LIN {X 0,Y 231.334,Z 988.847,A -85,B 0,C 180,E1 18236.93,E2 18236.93} C_VEL
LIN {X 0,Y 220.911,Z 1008.235,A -85,B 0,C 180,E1 18251.991,E2 18251.991} C_VEL
LIN {X 0,Y 219.134,Z 1015.208,A -85,B 0,C 180,E1 18264.035,E2 18264.035} C_VEL
LIN {X 0,Y 219.137,Z 1015.4,A -85,B 0,C 180,E1 18275.961,E2 18275.961} C_VEL
LIN {X 0,Y 222.596,Z 1005.334,A -85,B 0,C 180,E1 18292.021,E2 18292.021} C_VEL
LIN {X 0,Y 238.295,Z 981.214,A -85,B 0,C 180,E1 18308.382,E2 18308.382} C_VEL
LIN {X 0,Y 267.201,Z 942.328,A -85,B 0,C 180,E1 18321.811,E2 18321.811} C_VEL
LIN {X 0,Y 301.641,Z 891.524,A -85,B 0,C 180,E1 18330.943,E2 18330.943} C_VEL
LIN {X 0,Y 323.469,Z 851.273,A -85,B 0,C 180,E1 18335.504,E2 18335.504} C_VEL
LIN {X 0,Y 324.253,Z 838.125,A -85,B 0,C 180,E1 18342.326,E2 18342.326} C_VEL
LIN {X 0,Y 323.893,Z 839.008,A -85,B 0,C 180,E1 18347.863,E2 18347.863} C_VEL
LIN {X 0,Y 321.358,Z 853.442,A -85,B 0,C 180,E1 18354.273,E2 18354.273} C_VEL
LIN {X 0,Y 299.51,Z 890.449,A -85,B 0,C 180,E1 18358.703,E2 18358.703} C_VEL
LIN {X 0,Y 278.664,Z 915.584,A -85,B 0,C 180,E1 18361.445,E2 18361.445} C_VEL
LIN {X 0,Y 245.109,Z 956.502,A -85,B 0,C 180,E1 18372.917,E2 18372.917} C_VEL
LIN {X 0,Y 221.401,Z 984.345,A -85,B 0,C 180,E1 18388.646,E2 18388.646} C_VEL
LIN {X 0,Y 212.14,Z 997.349,A -85,B 0,C 180,E1 18404.662,E2 18404.662} C_VEL
LIN {X 0,Y 209.736,Z 999.603,A -85,B 0,C 180,E1 18421.947,E2 18421.947} C_VEL
LIN {X 0,Y 214.542,Z 991.139,A -85,B 0,C 180,E1 18437.75,E2 18437.75} C_VEL
LIN {X 0,Y 229.062,Z 968.541,A -85,B 0,C 180,E1 18454.559,E2 18454.559} C_VEL
LIN {X 0,Y 254.848,Z 932.339,A -85,B 0,C 180,E1 18467.893,E2 18467.893} C_VEL
LIN {X 0,Y 284.972,Z 883.616,A -85,B 0,C 180,E1 18477.345,E2 18477.345} C_VEL
LIN {X 0,Y 301.612,Z 849.625,A -85,B 0,C 180,E1 18481.47,E2 18481.47} C_VEL
LIN {X 0,Y 294.558,Z 819.144,A -85,B 0,C 180,E1 18491.629,E2 18491.629} C_VEL
LIN {X 0,Y 285.95,Z 795.84,A -85,B 0,C 180,E1 18503.391,E2 18503.391} C_VEL
LIN {X 0,Y 280.392,Z 783.23,A -85,B 0,C 180,E1 18516.018,E2 18516.018} C_VEL
LIN {X 0,Y 280.562,Z 781.44,A -85,B 0,C 180,E1 18529.053,E2 18529.053} C_VEL
LIN {X 0,Y 284.564,Z 787.554,A -85,B 0,C 180,E1 18538.437,E2 18538.437} C_VEL
LIN {X 0,Y 293.059,Z 807.387,A -85,B 0,C 180,E1 18550.405,E2 18550.405} C_VEL
LIN {X 0,Y 302.403,Z 835.998,A -85,B 0,C 180,E1 18560.91,E2 18560.91} C_VEL
LIN {X 0,Y 304.622,Z 853.266,A -85,B 0,C 180,E1 18565.354,E2 18565.354} C_VEL
LIN {X 0,Y 275.554,Z 910.337,A -85,B 0,C 180,E1 18572.136,E2 18572.136} C_VEL
LIN {X 0,Y 245.448,Z 957.331,A -85,B 0,C 180,E1 18582.736,E2 18582.736} C_VEL
LIN {X 0,Y 222.895,Z 990.368,A -85,B 0,C 180,E1 18596.995,E2 18596.995} C_VEL
LIN {X 0,Y 212.514,Z 1009.322,A -85,B 0,C 180,E1 18613.202,E2 18613.202} C_VEL
LIN {X 0,Y 211.113,Z 1015.708,A -85,B 0,C 180,E1 18627.938,E2 18627.938} C_VEL
LIN {X 0,Y 211.662,Z 1012.771,A -85,B 0,C 180,E1 18642.419,E2 18642.419} C_VEL
LIN {X 0,Y 220.362,Z 997.045,A -85,B 0,C 180,E1 18659.951,E2 18659.951} C_VEL
LIN {X 0,Y 244.359,Z 965.515,A -85,B 0,C 180,E1 18676.299,E2 18676.299} C_VEL
LIN {X 0,Y 278.974,Z 920.137,A -85,B 0,C 180,E1 18688.065,E2 18688.065} C_VEL
LIN {X 0,Y 314.593,Z 864.629,A -85,B 0,C 180,E1 18695.39,E2 18695.39} C_VEL
LIN {X 0,Y 319.046,Z 855.506,A -85,B 0,C 180,E1 18696.616,E2 18696.616} C_VEL
LIN {X 0,Y 320.141,Z 845.375,A -85,B 0,C 180,E1 18702.091,E2 18702.091} C_VEL
LIN {X 0,Y 319.7,Z 845.822,A -85,B 0,C 180,E1 18707.701,E2 18707.701} C_VEL
LIN {X 0,Y 316.504,Z 858.344,A -85,B 0,C 180,E1 18713.297,E2 18713.297} C_VEL
LIN {X 0,Y 281.686,Z 911.578,A -85,B 0,C 180,E1 18720.654,E2 18720.654} C_VEL
LIN {X 0,Y 278.664,Z 915.584,A -85,B 0,C 180,E1 18721.445,E2 18721.445} C_VEL
LIN {X 0,Y 256.83,Z 937.989,A -85,B 0,C 180,E1 18725.038,E2 18725.038} C_VEL
LIN {X 0,Y 224.568,Z 973.616,A -85,B 0,C 180,E1 18739.578,E2 18739.578} C_VEL
LIN {X 0,Y 207.548,Z 993.263,A -85,B 0,C 180,E1 18756.625,E2 18756.625} C_VEL
LIN {X 0,Y 201.91,Z 1000.154,A -85,B 0,C 180,E1 18772.174,E2 18772.174} C_VEL
LIN {X 0,Y 203.32,Z 997.547,A -85,B 0,C 180,E1 18789.01,E2 18789.01} C_VEL
LIN {X 0,Y 212.229,Z 982.956,A -85,B 0,C 180,E1 18806.501,E2 18806.501} C_VEL
LIN {X 0,Y 234.308,Z 953.213,A -85,B 0,C 180,E1 18822.646,E2 18822.646} C_VEL
LIN {X 0,Y 263.917,Z 910.873,A -85,B 0,C 180,E1 18834.188,E2 18834.188} C_VEL
LIN {X 0,Y 293.679,Z 858.461,A -85,B 0,C 180,E1 18841.767,E2 18841.767} C_VEL
LIN {X 0,Y 295.528,Z 850.294,A -85,B 0,C 180,E1 18843.304,E2 18843.304} C_VEL
LIN {X 0,Y 288.868,Z 821.3,A -85,B 0,C 180,E1 18853.805,E2 18853.805} C_VEL
LIN {X 0,Y 281.434,Z 800.636,A -85,B 0,C 180,E1 18865.481,E2 18865.481} C_VEL
LIN {X 0,Y 277.598,Z 790.868,A -85,B 0,C 180,E1 18875.761,E2 18875.761} C_VEL
LIN {X 0,Y 277.86,Z 788.939,A -85,B 0,C 180,E1 18888.945,E2 18888.945} C_VEL
LIN {X 0,Y 281.599,Z 795.076,A -85,B 0,C 180,E1 18898.421,E2 18898.421} C_VEL
LIN {X 0,Y 289.554,Z 815.2,A -85,B 0,C 180,E1 18910.532,E2 18910.532} C_VEL
LIN {X 0,Y 297.985,Z 844.388,A -85,B 0,C 180,E1 18921.235,E2 18921.235} C_VEL
LIN {X 0,Y 299.184,Z 855.972,A -85,B 0,C 180,E1 18924.294,E2 18924.294} C_VEL
LIN {X 0,Y 269.29,Z 912.298,A -85,B 0,C 180,E1 18931.138,E2 18931.138} C_VEL
LIN {X 0,Y 237.95,Z 959.184,A -85,B 0,C 180,E1 18942.085,E2 18942.085} C_VEL
LIN {X 0,Y 213.687,Z 993.04,A -85,B 0,C 180,E1 18957.813,E2 18957.813} C_VEL
LIN {X 0,Y 204.098,Z 1010.58,A -85,B 0,C 180,E1 18974.913,E2 18974.913} C_VEL
LIN {X 0,Y 203.112,Z 1015.397,A -85,B 0,C 180,E1 18987.857,E2 18987.857} C_VEL
LIN {X 0,Y 203.722,Z 1012.51,A -85,B 0,C 180,E1 19002.912,E2 19002.912} C_VEL
LIN {X 0,Y 213.178,Z 996.923,A -85,B 0,C 180,E1 19021.065,E2 19021.065} C_VEL
LIN {X 0,Y 239.023,Z 965.172,A -85,B 0,C 180,E1 19037.934,E2 19037.934} C_VEL
LIN {X 0,Y 275.499,Z 919.867,A -85,B 0,C 180,E1 19049.671,E2 19049.671} C_VEL
LIN {X 0,Y 312.833,Z 863.926,A -85,B 0,C 180,E1 19056.911,E2 19056.911} C_VEL
LIN {X 0,Y 315.38,Z 855.567,A -85,B 0,C 180,E1 19059.769,E2 19059.769} C_VEL
LIN {X 0,Y 316.057,Z 850.77,A -85,B 0,C 180,E1 19064.724,E2 19064.724} C_VEL
LIN {X 0,Y 313.716,Z 858.36,A -85,B 0,C 180,E1 19070.858,E2 19070.858} C_VEL
LIN {X 0,Y 310.109,Z 866.089,A -85,B 0,C 180,E1 19072.588,E2 19072.588} C_VEL
LIN {X 0,Y 273.08,Z 918.562,A -85,B 0,C 180,E1 19080.396,E2 19080.396} C_VEL
LIN {X 0,Y 256.83,Z 937.989,A -85,B 0,C 180,E1 19085.038,E2 19085.038} C_VEL
LIN {X 0,Y 234.754,Z 957.261,A -85,B 0,C 180,E1 19089.71,E2 19089.71} C_VEL
LIN {X 0,Y 206.942,Z 985.713,A -85,B 0,C 180,E1 19106.686,E2 19106.686} C_VEL
LIN {X 0,Y 196.73,Z 997.789,A -85,B 0,C 180,E1 19122.878,E2 19122.878} C_VEL
LIN {X 0,Y 193.391,Z 1000.578,A -85,B 0,C 180,E1 19139.334,E2 19139.334} C_VEL
LIN {X 0,Y 197.092,Z 995.113,A -85,B 0,C 180,E1 19154.396,E2 19154.396} C_VEL
LIN {X 0,Y 210.213,Z 975.921,A -85,B 0,C 180,E1 19172.796,E2 19172.796} C_VEL
LIN {X 0,Y 236.373,Z 942.604,A -85,B 0,C 180,E1 19187.758,E2 19187.758} C_VEL
LIN {X 0,Y 268.795,Z 895.644,A -85,B 0,C 180,E1 19198.361,E2 19198.361} C_VEL
LIN {X 0,Y 290.059,Z 855.543,A -85,B 0,C 180,E1 19203.794,E2 19203.794} C_VEL
LIN {X 0,Y 284.641,Z 828.293,A -85,B 0,C 180,E1 19213.929,E2 19213.929} C_VEL
LIN {X 0,Y 278.283,Z 808.54,A -85,B 0,C 180,E1 19225.034,E2 19225.034} C_VEL
LIN {X 0,Y 274.609,Z 798.301,A -85,B 0,C 180,E1 19235.766,E2 19235.766} C_VEL
LIN {X 0,Y 274.847,Z 796.329,A -85,B 0,C 180,E1 19248.823,E2 19248.823} C_VEL
LIN {X 0,Y 278.524,Z 802.579,A -85,B 0,C 180,E1 19258.403,E2 19258.403} C_VEL
LIN {X 0,Y 285.889,Z 822.963,A -85,B 0,C 180,E1 19270.669,E2 19270.669} C_VEL
LIN {X 0,Y 293.137,Z 851.47,A -85,B 0,C 180,E1 19281.205,E2 19281.205} C_VEL
LIN {X 0,Y 293.003,Z 860.497,A -85,B 0,C 180,E1 19283.349,E2 19283.349} C_VEL
LIN {X 0,Y 261.861,Z 916.194,A -85,B 0,C 180,E1 19290.447,E2 19290.447} C_VEL
LIN {X 0,Y 230.34,Z 961.065,A -85,B 0,C 180,E1 19301.456,E2 19301.456} C_VEL
LIN {X 0,Y 205.706,Z 993.851,A -85,B 0,C 180,E1 19317.53,E2 19317.53} C_VEL
LIN {X 0,Y 196.04,Z 1010.665,A -85,B 0,C 180,E1 19335.132,E2 19335.132} C_VEL
LIN {X 0,Y 195.102,Z 1015.084,A -85,B 0,C 180,E1 19347.769,E2 19347.769} C_VEL
LIN {X 0,Y 195.489,Z 1013.207,A -85,B 0,C 180,E1 19361.189,E2 19361.189} C_VEL
LIN {X 0,Y 204.554,Z 998.694,A -85,B 0,C 180,E1 19380.637,E2 19380.637} C_VEL
LIN {X 0,Y 231.069,Z 968.126,A -85,B 0,C 180,E1 19398.335,E2 19398.335} C_VEL
LIN {X 0,Y 268.675,Z 924.229,A -85,B 0,C 180,E1 19410.484,E2 19410.484} C_VEL
LIN {X 0,Y 308.422,Z 868.26,A -85,B 0,C 180,E1 19418.016,E2 19418.016} C_VEL
LIN {X 0,Y 310.955,Z 861.059,A -85,B 0,C 180,E1 19420.601,E2 19420.601} C_VEL
LIN {X 0,Y 311.637,Z 857.651,A -85,B 0,C 180,E1 19424.502,E2 19424.502} C_VEL
LIN {X 0,Y 309.306,Z 863.877,A -85,B 0,C 180,E1 19430.147,E2 19430.147} C_VEL
LIN {X 0,Y 304.024,Z 872.927,A -85,B 0,C 180,E1 19431.784,E2 19431.784} C_VEL
LIN {X 0,Y 265.573,Z 923.791,A -85,B 0,C 180,E1 19439.791,E2 19439.791} C_VEL
LIN {X 0,Y 234.754,Z 957.261,A -85,B 0,C 180,E1 19449.71,E2 19449.71} C_VEL
LIN {X 0,Y 213.753,Z 973.272,A -85,B 0,C 180,E1 19455.789,E2 19455.789} C_VEL
LIN {X 0,Y 192.855,Z 993.797,A -85,B 0,C 180,E1 19474.288,E2 19474.288} C_VEL
LIN {X 0,Y 185.769,Z 1000.904,A -85,B 0,C 180,E1 19492.218,E2 19492.218} C_VEL
LIN {X 0,Y 187.915,Z 997.347,A -85,B 0,C 180,E1 19511.315,E2 19511.315} C_VEL
LIN {X 0,Y 199.177,Z 981.483,A -85,B 0,C 180,E1 19530.074,E2 19530.074} C_VEL
LIN {X 0,Y 223.883,Z 951.382,A -85,B 0,C 180,E1 19546.239,E2 19546.239} C_VEL
LIN {X 0,Y 256.545,Z 907.703,A -85,B 0,C 180,E1 19557.741,E2 19557.741} C_VEL
LIN {X 0,Y 284.491,Z 860.005,A -85,B 0,C 180,E1 19564.548,E2 19564.548} C_VEL
LIN {X 0,Y 279.831,Z 833.495,A -85,B 0,C 180,E1 19574.829,E2 19574.829} C_VEL
LIN {X 0,Y 273.829,Z 813.189,A -85,B 0,C 180,E1 19587.258,E2 19587.258} C_VEL
LIN {X 0,Y 270.884,Z 804.65,A -85,B 0,C 180,E1 19598.61,E2 19598.61} C_VEL
LIN {X 0,Y 271.782,Z 803.697,A -85,B 0,C 180,E1 19608.695,E2 19608.695} C_VEL
LIN {X 0,Y 275.188,Z 809.94,A -85,B 0,C 180,E1 19618.384,E2 19618.384} C_VEL
LIN {X 0,Y 281.542,Z 828.995,A -85,B 0,C 180,E1 19630.051,E2 19630.051} C_VEL
LIN {X 0,Y 287.77,Z 856.236,A -85,B 0,C 180,E1 19640.475,E2 19640.475} C_VEL
LIN {X 0,Y 287.09,Z 864.112,A -85,B 0,C 180,E1 19642.317,E2 19642.317} C_VEL
LIN {X 0,Y 255.032,Z 919.161,A -85,B 0,C 180,E1 19649.544,E2 19649.544} C_VEL
LIN {X 0,Y 221.372,Z 964.645,A -85,B 0,C 180,E1 19661.383,E2 19661.383} C_VEL
LIN {X 0,Y 197.966,Z 994.244,A -85,B 0,C 180,E1 19676.961,E2 19676.961} C_VEL
LIN {X 0,Y 188.343,Z 1009.805,A -85,B 0,C 180,E1 19693.617,E2 19693.617} C_VEL
LIN {X 0,Y 187.101,Z 1014.772,A -85,B 0,C 180,E1 19707.674,E2 19707.674} C_VEL
LIN {X 0,Y 187.794,Z 1012.243,A -85,B 0,C 180,E1 19723.426,E2 19723.426} C_VEL
LIN {X 0,Y 198.733,Z 997.113,A -85,B 0,C 180,E1 19743.214,E2 19743.214} C_VEL
LIN {X 0,Y 228.688,Z 965.09,A -85,B 0,C 180,E1 19761.218,E2 19761.218} C_VEL
LIN {X 0,Y 268.565,Z 920.5,A -85,B 0,C 180,E1 19772.833,E2 19772.833} C_VEL
LIN {X 0,Y 305.757,Z 869.649,A -85,B 0,C 180,E1 19779.653,E2 19779.653} C_VEL
LIN {X 0,Y 307.096,Z 864.294,A -85,B 0,C 180,E1 19784.498,E2 19784.498} C_VEL
LIN {X 0,Y 304.96,Z 868.97,A -85,B 0,C 180,E1 19789.258,E2 19789.258} C_VEL
LIN {X 0,Y 297.61,Z 880.195,A -85,B 0,C 180,E1 19791.023,E2 19791.023} C_VEL
LIN {X 0,Y 257.04,Z 930.122,A -85,B 0,C 180,E1 19799.425,E2 19799.425} C_VEL
LIN {X 0,Y 220.352,Z 966.958,A -85,B 0,C 180,E1 19812.265,E2 19812.265} C_VEL
LIN {X 0,Y 213.753,Z 973.272,A -85,B 0,C 180,E1 19815.789,E2 19815.789} C_VEL
LIN {X 0,Y 194.068,Z 985.971,A -85,B 0,C 180,E1 19823.301,E2 19823.301} C_VEL
LIN {X 0,Y 181.379,Z 998.29,A -85,B 0,C 180,E1 19840.815,E2 19840.815} C_VEL
LIN {X 0,Y 177.298,Z 1001.434,A -85,B 0,C 180,E1 19856.197,E2 19856.197} C_VEL
LIN {X 0,Y 181.076,Z 996.118,A -85,B 0,C 180,E1 19874.697,E2 19874.697} C_VEL
LIN {X 0,Y 195.447,Z 977.515,A -85,B 0,C 180,E1 19894.455,E2 19894.455} C_VEL
LIN {X 0,Y 224.171,Z 944.246,A -85,B 0,C 180,E1 19910.303,E2 19910.303} C_VEL
LIN {X 0,Y 258.34,Z 898.219,A -85,B 0,C 180,E1 19920.933,E2 19920.933} C_VEL
LIN {X 0,Y 278.842,Z 863.563,A -85,B 0,C 180,E1 19925.614,E2 19925.614} C_VEL
LIN {X 0,Y 274.781,Z 837.593,A -85,B 0,C 180,E1 19936.304,E2 19936.304} C_VEL
LIN {X 0,Y 269.524,Z 818.372,A -85,B 0,C 180,E1 19949.094,E2 19949.094} C_VEL
LIN {X 0,Y 267.535,Z 810.942,A -85,B 0,C 180,E1 19961.786,E2 19961.786} C_VEL
LIN {X 0,Y 270.733,Z 813.68,A -85,B 0,C 180,E1 19975.141,E2 19975.141} C_VEL
LIN {X 0,Y 276.265,Z 831.85,A -85,B 0,C 180,E1 19987.855,E2 19987.855} C_VEL
LIN {X 0,Y 281.999,Z 858.161,A -85,B 0,C 180,E1 19998.797,E2 19998.797} C_VEL
LIN {X 0,Y 281.654,Z 866.97,A -85,B 0,C 180,E1 20001.181,E2 20001.181} C_VEL
LIN {X 0,Y 248.416,Z 921.576,A -85,B 0,C 180,E1 20008.532,E2 20008.532} C_VEL
LIN {X 0,Y 213.941,Z 966.197,A -85,B 0,C 180,E1 20020.582,E2 20020.582} C_VEL
LIN {X 0,Y 189.581,Z 995.518,A -85,B 0,C 180,E1 20037.076,E2 20037.076} C_VEL
LIN {X 0,Y 179.86,Z 1010.863,A -85,B 0,C 180,E1 20055.722,E2 20055.722} C_VEL
LIN {X 0,Y 179.265,Z 1014.624,A -85,B 0,C 180,E1 20072.424,E2 20072.424} C_VEL
LIN {X 0,Y 182.356,Z 1007.925,A -85,B 0,C 180,E1 20091.991,E2 20091.991} C_VEL
LIN {X 0,Y 202.001,Z 986.423,A -85,B 0,C 180,E1 20112.541,E2 20112.541} C_VEL
LIN {X 0,Y 238.624,Z 950.181,A -85,B 0,C 180,E1 20127.893,E2 20127.893} C_VEL
LIN {X 0,Y 281.051,Z 902.165,A -85,B 0,C 180,E1 20137.356,E2 20137.356} C_VEL
LIN {X 0,Y 301.377,Z 874.097,A -85,B 0,C 180,E1 20140.935,E2 20140.935} C_VEL
LIN {X 0,Y 302.26,Z 871.131,A -85,B 0,C 180,E1 20144.008,E2 20144.008} C_VEL
LIN {X 0,Y 300.248,Z 874.828,A -85,B 0,C 180,E1 20148.707,E2 20148.707} C_VEL
LIN {X 0,Y 257.072,Z 927.132,A -85,B 0,C 180,E1 20156.896,E2 20156.896} C_VEL
LIN {X 0,Y 217.472,Z 965.308,A -85,B 0,C 180,E1 20169.432,E2 20169.432} C_VEL
LIN {X 0,Y 194.068,Z 985.971,A -85,B 0,C 180,E1 20183.301,E2 20183.301} C_VEL
LIN {X 0,Y 177.681,Z 995.01,A -85,B 0,C 180,E1 20192.644,E2 20192.644} C_VEL
LIN {X 0,Y 170.288,Z 1001.234,A -85,B 0,C 180,E1 20209.32,E2 20209.32} C_VEL
LIN {X 0,Y 170.976,Z 999.243,A -85,B 0,C 180,E1 20228.873,E2 20228.873} C_VEL
LIN {X 0,Y 180.284,Z 987.222,A -85,B 0,C 180,E1 20247.59,E2 20247.59} C_VEL
LIN {X 0,Y 204.97,Z 959.987,A -85,B 0,C 180,E1 20265.896,E2 20265.896} C_VEL
LIN {X 0,Y 239.725,Z 918.482,A -85,B 0,C 180,E1 20278.729,E2 20278.729} C_VEL
LIN {X 0,Y 273.111,Z 866.658,A -85,B 0,C 180,E1 20286.875,E2 20286.875} C_VEL
LIN {X 0,Y 269.766,Z 841.862,A -85,B 0,C 180,E1 20297.697,E2 20297.697} C_VEL
LIN {X 0,Y 265.842,Z 825.629,A -85,B 0,C 180,E1 20309.049,E2 20309.049} C_VEL
LIN {X 0,Y 264.085,Z 818.263,A -85,B 0,C 180,E1 20321.54,E2 20321.54} C_VEL
LIN {X 0,Y 267.167,Z 820.932,A -85,B 0,C 180,E1 20335.076,E2 20335.076} C_VEL
LIN {X 0,Y 272.113,Z 839.271,A -85,B 0,C 180,E1 20347.975,E2 20347.975} C_VEL
LIN {X 0,Y 276.785,Z 864.323,A -85,B 0,C 180,E1 20358.542,E2 20358.542} C_VEL
LIN {X 0,Y 275.65,Z 870.987,A -85,B 0,C 180,E1 20360.118,E2 20360.118} C_VEL
LIN {X 0,Y 241.565,Z 924.41,A -85,B 0,C 180,E1 20367.566,E2 20367.566} C_VEL
LIN {X 0,Y 206.832,Z 967.314,A -85,B 0,C 180,E1 20379.605,E2 20379.605} C_VEL
LIN {X 0,Y 181.322,Z 996.586,A -85,B 0,C 180,E1 20397.039,E2 20397.039} C_VEL
LIN {X 0,Y 171.63,Z 1011.484,A -85,B 0,C 180,E1 20417.227,E2 20417.227} C_VEL
LIN {X 0,Y 171.264,Z 1014.334,A -85,B 0,C 180,E1 20432.537,E2 20432.537} C_VEL
LIN {X 0,Y 173.734,Z 1009.157,A -85,B 0,C 180,E1 20450.449,E2 20450.449} C_VEL
LIN {X 0,Y 192.553,Z 989.611,A -85,B 0,C 180,E1 20472.058,E2 20472.058} C_VEL
LIN {X 0,Y 230.455,Z 954.665,A -85,B 0,C 180,E1 20488.436,E2 20488.436} C_VEL
LIN {X 0,Y 275.41,Z 906.835,A -85,B 0,C 180,E1 20498.41,E2 20498.41} C_VEL
LIN {X 0,Y 296.027,Z 880.706,A -85,B 0,C 180,E1 20501.511,E2 20501.511} C_VEL
LIN {X 0,Y 297.336,Z 877.785,A -85,B 0,C 180,E1 20503.736,E2 20503.736} C_VEL
LIN {X 0,Y 295.38,Z 880.557,A -85,B 0,C 180,E1 20507.766,E2 20507.766} C_VEL
LIN {X 0,Y 251.053,Z 931.031,A -85,B 0,C 180,E1 20515.854,E2 20515.854} C_VEL
LIN {X 0,Y 209.872,Z 968.156,A -85,B 0,C 180,E1 20528.782,E2 20528.782} C_VEL
LIN {X 0,Y 180.971,Z 992.098,A -85,B 0,C 180,E1 20548.301,E2 20548.301} C_VEL
LIN {X 0,Y 177.681,Z 995.01,A -85,B 0,C 180,E1 20552.644,E2 20552.644} C_VEL
LIN {X 0,Y 163.943,Z 1000.518,A -85,B 0,C 180,E1 20563.553,E2 20563.553} C_VEL
LIN {X 0,Y 161.896,Z 1000.774,A -85,B 0,C 180,E1 20585.053,E2 20585.053} C_VEL
LIN {X 0,Y 169.187,Z 991.814,A -85,B 0,C 180,E1 20603.565,E2 20603.565} C_VEL
LIN {X 0,Y 191.6,Z 967.799,A -85,B 0,C 180,E1 20623.748,E2 20623.748} C_VEL
LIN {X 0,Y 226.625,Z 929.183,A -85,B 0,C 180,E1 20637.955,E2 20637.955} C_VEL
LIN {X 0,Y 262.917,Z 878.68,A -85,B 0,C 180,E1 20646.79,E2 20646.79} C_VEL
LIN {X 0,Y 267.437,Z 869.992,A -85,B 0,C 180,E1 20648.118,E2 20648.118} C_VEL
LIN {X 0,Y 264.863,Z 846.938,A -85,B 0,C 180,E1 20658.744,E2 20658.744} C_VEL
LIN {X 0,Y 261.578,Z 831.468,A -85,B 0,C 180,E1 20670.416,E2 20670.416} C_VEL
LIN {X 0,Y 260.796,Z 824.922,A -85,B 0,C 180,E1 20684.783,E2 20684.783} C_VEL
LIN {X 0,Y 264.03,Z 830.528,A -85,B 0,C 180,E1 20697.272,E2 20697.272} C_VEL
LIN {X 0,Y 268.191,Z 848.196,A -85,B 0,C 180,E1 20708.912,E2 20708.912} C_VEL
LIN {X 0,Y 271.553,Z 871.209,A -85,B 0,C 180,E1 20718.559,E2 20718.559} C_VEL
LIN {X 0,Y 236.131,Z 925.362,A -85,B 0,C 180,E1 20726.177,E2 20726.177} C_VEL
LIN {X 0,Y 200.478,Z 967.64,A -85,B 0,C 180,E1 20738.242,E2 20738.242} C_VEL
LIN {X 0,Y 174.189,Z 996.225,A -85,B 0,C 180,E1 20755.737,E2 20755.737} C_VEL
LIN {X 0,Y 163.696,Z 1011.097,A -85,B 0,C 180,E1 20776.596,E2 20776.596} C_VEL
LIN {X 0,Y 163.238,Z 1014.045,A -85,B 0,C 180,E1 20792.662,E2 20792.662} C_VEL
LIN {X 0,Y 166.022,Z 1008.958,A -85,B 0,C 180,E1 20811.444,E2 20811.444} C_VEL
LIN {X 0,Y 186.464,Z 989.689,A -85,B 0,C 180,E1 20833.77,E2 20833.77} C_VEL
LIN {X 0,Y 227.416,Z 954.19,A -85,B 0,C 180,E1 20850.531,E2 20850.531} C_VEL
LIN {X 0,Y 274.407,Z 906.262,A -85,B 0,C 180,E1 20860.232,E2 20860.232} C_VEL
LIN {X 0,Y 292.081,Z 884.634,A -85,B 0,C 180,E1 20863.02,E2 20863.02} C_VEL
LIN {X 0,Y 290.823,Z 885.772,A -85,B 0,C 180,E1 20866.662,E2 20866.662} C_VEL
LIN {X 0,Y 245.291,Z 934.54,A -85,B 0,C 180,E1 20874.718,E2 20874.718} C_VEL
LIN {X 0,Y 201.905,Z 971.275,A -85,B 0,C 180,E1 20888.253,E2 20888.253} C_VEL
LIN {X 0,Y 172.177,Z 994.121,A -85,B 0,C 180,E1 20909.057,E2 20909.057} C_VEL
LIN {X 0,Y 163.943,Z 1000.518,A -85,B 0,C 180,E1 20923.553,E2 20923.553} C_VEL
LIN {X 0,Y 153.147,Z 1002.217,A -85,B 0,C 180,E1 20935.814,E2 20935.814} C_VEL
LIN {X 0,Y 157.374,Z 997.193,A -85,B 0,C 180,E1 20956.052,E2 20956.052} C_VEL
LIN {X 0,Y 173.69,Z 979.697,A -85,B 0,C 180,E1 20977.533,E2 20977.533} C_VEL
LIN {X 0,Y 207.085,Z 946.127,A -85,B 0,C 180,E1 20994.79,E2 20994.79} C_VEL
LIN {X 0,Y 245.278,Z 899.528,A -85,B 0,C 180,E1 21005.541,E2 21005.541} C_VEL
LIN {X 0,Y 261.881,Z 874.141,A -85,B 0,C 180,E1 21009.078,E2 21009.078} C_VEL
LIN {X 0,Y 259.937,Z 851.575,A -85,B 0,C 180,E1 21020.106,E2 21020.106} C_VEL
LIN {X 0,Y 257.301,Z 837.302,A -85,B 0,C 180,E1 21031.809,E2 21031.809} C_VEL
LIN {X 0,Y 257.023,Z 832.026,A -85,B 0,C 180,E1 21044.555,E2 21044.555} C_VEL
LIN {X 0,Y 259.849,Z 836.881,A -85,B 0,C 180,E1 21056.614,E2 21056.614} C_VEL
LIN {X 0,Y 263.379,Z 853.873,A -85,B 0,C 180,E1 21068.242,E2 21068.242} C_VEL
LIN {X 0,Y 265.907,Z 874.525,A -85,B 0,C 180,E1 21077.33,E2 21077.33} C_VEL
LIN {X 0,Y 228.668,Z 929.082,A -85,B 0,C 180,E1 21085.274,E2 21085.274} C_VEL
LIN {X 0,Y 190.934,Z 971.401,A -85,B 0,C 180,E1 21098.286,E2 21098.286} C_VEL
LIN {X 0,Y 164.911,Z 998.297,A -85,B 0,C 180,E1 21116.795,E2 21116.795} C_VEL
LIN {X 0,Y 155.806,Z 1010.689,A -85,B 0,C 180,E1 21135.904,E2 21135.904} C_VEL
LIN {X 0,Y 155.211,Z 1013.754,A -85,B 0,C 180,E1 21152.8,E2 21152.8} C_VEL
LIN {X 0,Y 158.367,Z 1008.771,A -85,B 0,C 180,E1 21172.536,E2 21172.536} C_VEL
LIN {X 0,Y 180.539,Z 989.796,A -85,B 0,C 180,E1 21195.599,E2 21195.599} C_VEL
LIN {X 0,Y 224.39,Z 954.076,A -85,B 0,C 180,E1 21212.578,E2 21212.578} C_VEL
LIN {X 0,Y 272.74,Z 906.901,A -85,B 0,C 180,E1 21221.914,E2 21221.914} C_VEL
LIN {X 0,Y 287.069,Z 890.322,A -85,B 0,C 180,E1 21224.218,E2 21224.218} C_VEL
LIN {X 0,Y 285.687,Z 891.829,A -85,B 0,C 180,E1 21225.621,E2 21225.621} C_VEL
LIN {X 0,Y 237.414,Z 940.054,A -85,B 0,C 180,E1 21234.017,E2 21234.017} C_VEL
LIN {X 0,Y 191.875,Z 975.721,A -85,B 0,C 180,E1 21248.651,E2 21248.651} C_VEL
LIN {X 0,Y 162.525,Z 996.445,A -85,B 0,C 180,E1 21270.965,E2 21270.965} C_VEL
LIN {X 0,Y 153.916,Z 1002.167,A -85,B 0,C 180,E1 21290.145,E2 21290.145} C_VEL
LIN {X 0,Y 153.147,Z 1002.217,A -85,B 0,C 180,E1 21295.814,E2 21295.814} C_VEL
LIN {X 0,Y 146.77,Z 1000.324,A -85,B 0,C 180,E1 21309.188,E2 21309.188} C_VEL
LIN {X 0,Y 157.429,Z 989.105,A -85,B 0,C 180,E1 21329.976,E2 21329.976} C_VEL
LIN {X 0,Y 186.783,Z 961.548,A -85,B 0,C 180,E1 21350.483,E2 21350.483} C_VEL
LIN {X 0,Y 226.05,Z 919.513,A -85,B 0,C 180,E1 21363.635,E2 21363.635} C_VEL
LIN {X 0,Y 256.267,Z 877.611,A -85,B 0,C 180,E1 21370.31,E2 21370.31} C_VEL
LIN {X 0,Y 254.9,Z 856.544,A -85,B 0,C 180,E1 21381.269,E2 21381.269} C_VEL
LIN {X 0,Y 253.05,Z 843.144,A -85,B 0,C 180,E1 21393.232,E2 21393.232} C_VEL
LIN {X 0,Y 253.05,Z 839.058,A -85,B 0,C 180,E1 21404.306,E2 21404.306} C_VEL
LIN {X 0,Y 255.802,Z 843.878,A -85,B 0,C 180,E1 21416.56,E2 21416.56} C_VEL
LIN {X 0,Y 258.763,Z 861.017,A -85,B 0,C 180,E1 21428.39,E2 21428.39} C_VEL
LIN {X 0,Y 259.779,Z 879.234,A -85,B 0,C 180,E1 21436.355,E2 21436.355} C_VEL
LIN {X 0,Y 222.765,Z 930.677,A -85,B 0,C 180,E1 21443.924,E2 21443.924} C_VEL
LIN {X 0,Y 183.578,Z 972.771,A -85,B 0,C 180,E1 21457.278,E2 21457.278} C_VEL
LIN {X 0,Y 155.941,Z 999.921,A -85,B 0,C 180,E1 21477.636,E2 21477.636} C_VEL
LIN {X 0,Y 147.115,Z 1012.091,A -85,B 0,C 180,E1 21501.096,E2 21501.096} C_VEL
LIN {X 0,Y 147.113,Z 1012.965,A -85,B 0,C 180,E1 21518.899,E2 21518.899} C_VEL
LIN {X 0,Y 156.231,Z 1003.989,A -85,B 0,C 180,E1 21542.291,E2 21542.291} C_VEL
LIN {X 0,Y 190.312,Z 978.576,A -85,B 0,C 180,E1 21564.817,E2 21564.817} C_VEL
LIN {X 0,Y 238.714,Z 939.313,A -85,B 0,C 180,E1 21578.394,E2 21578.394} C_VEL
LIN {X 0,Y 278.518,Z 899.892,A -85,B 0,C 180,E1 21584.546,E2 21584.546} C_VEL
LIN {X 0,Y 226.273,Z 947.876,A -85,B 0,C 180,E1 21593.996,E2 21593.996} C_VEL
LIN {X 0,Y 181.644,Z 979.927,A -85,B 0,C 180,E1 21609.142,E2 21609.142} C_VEL
LIN {X 0,Y 153.216,Z 998.365,A -85,B 0,C 180,E1 21632.661,E2 21632.661} C_VEL
LIN {X 0,Y 145.09,Z 1002.591,A -85,B 0,C 180,E1 21655.702,E2 21655.702} C_VEL
LIN {X 0,Y 146.77,Z 1000.324,A -85,B 0,C 180,E1 21669.188,E2 21669.188} C_VEL
LIN {X 0,Y 144.402,Z 994.947,A -85,B 0,C 180,E1 21683.079,E2 21683.079} C_VEL
LIN {X 0,Y 167.916,Z 973.548,A -85,B 0,C 180,E1 21705.734,E2 21705.734} C_VEL
LIN {X 0,Y 205.981,Z 937.39,A -85,B 0,C 180,E1 21721.215,E2 21721.215} C_VEL
LIN {X 0,Y 246.556,Z 887.777,A -85,B 0,C 180,E1 21730.592,E2 21730.592} C_VEL
LIN {X 0,Y 250.742,Z 880.052,A -85,B 0,C 180,E1 21732.046,E2 21732.046} C_VEL
LIN {X 0,Y 249.779,Z 859.678,A -85,B 0,C 180,E1 21743.76,E2 21743.76} C_VEL
LIN {X 0,Y 248.604,Z 849.213,A -85,B 0,C 180,E1 21754.533,E2 21754.533} C_VEL
LIN {X 0,Y 249.5,Z 846.162,A -85,B 0,C 180,E1 21767.67,E2 21767.67} C_VEL
LIN {X 0,Y 251.765,Z 852.591,A -85,B 0,C 180,E1 21778.233,E2 21778.233} C_VEL
LIN {X 0,Y 254.276,Z 871.775,A -85,B 0,C 180,E1 21790.444,E2 21790.444} C_VEL
LIN {X 0,Y 253.467,Z 883.768,A -85,B 0,C 180,E1 21795.169,E2 21795.169} C_VEL
LIN {X 0,Y 213.601,Z 936.151,A -85,B 0,C 180,E1 21803.363,E2 21803.363} C_VEL
LIN {X 0,Y 174.043,Z 976.122,A -85,B 0,C 180,E1 21817.308,E2 21817.308} C_VEL
LIN {X 0,Y 146.827,Z 1001.625,A -85,B 0,C 180,E1 21838.879,E2 21838.879} C_VEL
LIN {X 0,Y 139.154,Z 1011.695,A -85,B 0,C 180,E1 21860.582,E2 21860.582} C_VEL
LIN {X 0,Y 139.156,Z 1012.677,A -85,B 0,C 180,E1 21879.412,E2 21879.412} C_VEL
LIN {X 0,Y 151.117,Z 1002.583,A -85,B 0,C 180,E1 21905.966,E2 21905.966} C_VEL
LIN {X 0,Y 188.116,Z 977.188,A -85,B 0,C 180,E1 21927.89,E2 21927.89} C_VEL
LIN {X 0,Y 240.546,Z 936.436,A -85,B 0,C 180,E1 21941.031,E2 21941.031} C_VEL
LIN {X 0,Y 264.985,Z 913.838,A -85,B 0,C 180,E1 21944.824,E2 21944.824} C_VEL
LIN {X 0,Y 212.866,Z 956.758,A -85,B 0,C 180,E1 21954.528,E2 21954.528} C_VEL
LIN {X 0,Y 167.783,Z 985.938,A -85,B 0,C 180,E1 21971.561,E2 21971.561} C_VEL
LIN {X 0,Y 142.553,Z 1000.753,A -85,B 0,C 180,E1 21997.024,E2 21997.024} C_VEL
LIN {X 0,Y 137.093,Z 1002.569,A -85,B 0,C 180,E1 22020.126,E2 22020.126} C_VEL
LIN {X 0,Y 144.402,Z 994.947,A -85,B 0,C 180,E1 22043.079,E2 22043.079} C_VEL
LIN {X 0,Y 147.008,Z 986.464,A -85,B 0,C 180,E1 22056.653,E2 22056.653} C_VEL
LIN {X 0,Y 181.916,Z 956.572,A -85,B 0,C 180,E1 22076.671,E2 22076.671} C_VEL
LIN {X 0,Y 222.303,Z 914.776,A -85,B 0,C 180,E1 22088.218,E2 22088.218} C_VEL
LIN {X 0,Y 245.132,Z 885.142,A -85,B 0,C 180,E1 22092.646,E2 22092.646} C_VEL
LIN {X 0,Y 244.992,Z 866.148,A -85,B 0,C 180,E1 22103.911,E2 22103.911} C_VEL
LIN {X 0,Y 244.234,Z 855.113,A -85,B 0,C 180,E1 22116.14,E2 22116.14} C_VEL
LIN {X 0,Y 245.225,Z 852.942,A -85,B 0,C 180,E1 22127.452,E2 22127.452} C_VEL
LIN {X 0,Y 247.287,Z 859.389,A -85,B 0,C 180,E1 22138.201,E2 22138.201} C_VEL
LIN {X 0,Y 248.984,Z 877.707,A -85,B 0,C 180,E1 22150.135,E2 22150.135} C_VEL
LIN {X 0,Y 248.355,Z 886.343,A -85,B 0,C 180,E1 22153.774,E2 22153.774} C_VEL
LIN {X 0,Y 207.166,Z 938.435,A -85,B 0,C 180,E1 22162.046,E2 22162.046} C_VEL
LIN {X 0,Y 166.644,Z 977.418,A -85,B 0,C 180,E1 22176.21,E2 22176.21} C_VEL
LIN {X 0,Y 138.709,Z 1002.1,A -85,B 0,C 180,E1 22198.685,E2 22198.685} C_VEL
LIN {X 0,Y 131.169,Z 1011.288,A -85,B 0,C 180,E1 22220.003,E2 22220.003} C_VEL
LIN {X 0,Y 131.174,Z 1012.388,A -85,B 0,C 180,E1 22239.991,E2 22239.991} C_VEL
LIN {X 0,Y 142.503,Z 1003.797,A -85,B 0,C 180,E1 22265.851,E2 22265.851} C_VEL
LIN {X 0,Y 181.219,Z 979.288,A -85,B 0,C 180,E1 22289.13,E2 22289.13} C_VEL
LIN {X 0,Y 234.818,Z 940.359,A -85,B 0,C 180,E1 22302.314,E2 22302.314} C_VEL
LIN {X 0,Y 250.508,Z 927.008,A -85,B 0,C 180,E1 22304.908,E2 22304.908} C_VEL
LIN {X 0,Y 197.371,Z 966.078,A -85,B 0,C 180,E1 22315.658,E2 22315.658} C_VEL
LIN {X 0,Y 154.24,Z 991.032,A -85,B 0,C 180,E1 22334.303,E2 22334.303} C_VEL
LIN {X 0,Y 133.381,Z 1001.907,A -85,B 0,C 180,E1 22358.825,E2 22358.825} C_VEL
LIN {X 0,Y 129.766,Z 1001.904,A -85,B 0,C 180,E1 22385.841,E2 22385.841} C_VEL
LIN {X 0,Y 139.584,Z 992.684,A -85,B 0,C 180,E1 22408.445,E2 22408.445} C_VEL
LIN {X 0,Y 147.008,Z 986.464,A -85,B 0,C 180,E1 22416.653,E2 22416.653} C_VEL
LIN {X 0,Y 155.035,Z 974.872,A -85,B 0,C 180,E1 22429.055,E2 22429.055} C_VEL
LIN {X 0,Y 195.832,Z 939.301,A -85,B 0,C 180,E1 22444.683,E2 22444.683} C_VEL
LIN {X 0,Y 238.371,Z 890.346,A -85,B 0,C 180,E1 22453.788,E2 22453.788} C_VEL
LIN {X 0,Y 240.037,Z 874.97,A -85,B 0,C 180,E1 22462.216,E2 22462.216} C_VEL
LIN {X 0,Y 239.711,Z 863.121,A -85,B 0,C 180,E1 22473.747,E2 22473.747} C_VEL
LIN {X 0,Y 240.84,Z 859.656,A -85,B 0,C 180,E1 22487.614,E2 22487.614} C_VEL
LIN {X 0,Y 242.622,Z 866.026,A -85,B 0,C 180,E1 22498.167,E2 22498.167} C_VEL
LIN {X 0,Y 243.679,Z 883.624,A -85,B 0,C 180,E1 22509.814,E2 22509.814} C_VEL
LIN {X 0,Y 242.057,Z 890.754,A -85,B 0,C 180,E1 22512.535,E2 22512.535} C_VEL
LIN {X 0,Y 200.724,Z 940.611,A -85,B 0,C 180,E1 22520.665,E2 22520.665} C_VEL
LIN {X 0,Y 158.381,Z 979.41,A -85,B 0,C 180,E1 22535.461,E2 22535.461} C_VEL
LIN {X 0,Y 129.217,Z 1003.874,A -85,B 0,C 180,E1 22560.634,E2 22560.634} C_VEL
LIN {X 0,Y 122.977,Z 1012.063,A -85,B 0,C 180,E1 22586.459,E2 22586.459} C_VEL
LIN {X 0,Y 124.426,Z 1011.03,A -85,B 0,C 180,E1 22607.75,E2 22607.75} C_VEL
LIN {X 0,Y 145.543,Z 998.147,A -85,B 0,C 180,E1 22636.309,E2 22636.309} C_VEL
LIN {X 0,Y 195.012,Z 968.463,A -85,B 0,C 180,E1 22656.719,E2 22656.719} C_VEL
LIN {X 0,Y 236.214,Z 938.679,A -85,B 0,C 180,E1 22665.005,E2 22665.005} C_VEL
LIN {X 0,Y 182.746,Z 973.766,A -85,B 0,C 180,E1 22676.736,E2 22676.736} C_VEL
LIN {X 0,Y 140.379,Z 995.655,A -85,B 0,C 180,E1 22698.153,E2 22698.153} C_VEL
LIN {X 0,Y 123.641,Z 1003.05,A -85,B 0,C 180,E1 22722.558,E2 22722.558} C_VEL
LIN {X 0,Y 122.285,Z 1001.579,A -85,B 0,C 180,E1 22748.746,E2 22748.746} C_VEL
LIN {X 0,Y 134.985,Z 990.795,A -85,B 0,C 180,E1 22773.225,E2 22773.225} C_VEL
LIN {X 0,Y 155.035,Z 974.872,A -85,B 0,C 180,E1 22789.055,E2 22789.055} C_VEL
LIN {X 0,Y 168.442,Z 960.146,A -85,B 0,C 180,E1 22799.506,E2 22799.506} C_VEL
LIN {X 0,Y 212.124,Z 918.653,A -85,B 0,C 180,E1 22811.391,E2 22811.391} C_VEL
LIN {X 0,Y 234.106,Z 891.436,A -85,B 0,C 180,E1 22815.829,E2 22815.829} C_VEL
LIN {X 0,Y 234.98,Z 874.447,A -85,B 0,C 180,E1 22827.91,E2 22827.91} C_VEL
LIN {X 0,Y 235.171,Z 867.15,A -85,B 0,C 180,E1 22839.347,E2 22839.347} C_VEL
LIN {X 0,Y 237.227,Z 867.936,A -85,B 0,C 180,E1 22852.568,E2 22852.568} C_VEL
LIN {X 0,Y 238.153,Z 880.956,A -85,B 0,C 180,E1 22864.525,E2 22864.525} C_VEL
LIN {X 0,Y 237.492,Z 892.799,A -85,B 0,C 180,E1 22870.971,E2 22870.971} C_VEL
LIN {X 0,Y 194.752,Z 942.415,A -85,B 0,C 180,E1 22879.114,E2 22879.114} C_VEL
LIN {X 0,Y 153.645,Z 978.546,A -85,B 0,C 180,E1 22892.901,E2 22892.901} C_VEL
LIN {X 0,Y 123.539,Z 1001.971,A -85,B 0,C 180,E1 22916.437,E2 22916.437} C_VEL
LIN {X 0,Y 114.978,Z 1011.021,A -85,B 0,C 180,E1 22941.171,E2 22941.171} C_VEL
LIN {X 0,Y 115.268,Z 1011.816,A -85,B 0,C 180,E1 22961.386,E2 22961.386} C_VEL
LIN {X 0,Y 130.151,Z 1003.312,A -85,B 0,C 180,E1 22990.854,E2 22990.854} C_VEL
LIN {X 0,Y 176.181,Z 978.506,A -85,B 0,C 180,E1 23014.745,E2 23014.745} C_VEL
LIN {X 0,Y 221.192,Z 949.716,A -85,B 0,C 180,E1 23024.65,E2 23024.65} C_VEL
LIN {X 0,Y 164.137,Z 982.574,A -85,B 0,C 180,E1 23039.558,E2 23039.558} C_VEL
LIN {X 0,Y 125.288,Z 1000.054,A -85,B 0,C 180,E1 23065.166,E2 23065.166} C_VEL
LIN {X 0,Y 113.108,Z 1003.872,A -85,B 0,C 180,E1 23092.864,E2 23092.864} C_VEL
LIN {X 0,Y 117.777,Z 999.045,A -85,B 0,C 180,E1 23118.859,E2 23118.859} C_VEL
LIN {X 0,Y 140.334,Z 981.878,A -85,B 0,C 180,E1 23145.688,E2 23145.688} C_VEL
LIN {X 0,Y 168.442,Z 960.146,A -85,B 0,C 180,E1 23159.506,E2 23159.506} C_VEL
LIN {X 0,Y 184.614,Z 942.622,A -85,B 0,C 180,E1 23168.064,E2 23168.064} C_VEL
LIN {X 0,Y 227.781,Z 896.775,A -85,B 0,C 180,E1 23176.701,E2 23176.701} C_VEL
LIN {X 0,Y 229.707,Z 883.132,A -85,B 0,C 180,E1 23185.793,E2 23185.793} C_VEL
LIN {X 0,Y 230.119,Z 875.646,A -85,B 0,C 180,E1 23194.576,E2 23194.576} C_VEL
LIN {X 0,Y 231.366,Z 872.663,A -85,B 0,C 180,E1 23206.687,E2 23206.687} C_VEL
LIN {X 0,Y 232.775,Z 877.072,A -85,B 0,C 180,E1 23216.22,E2 23216.22} C_VEL
LIN {X 0,Y 232.637,Z 893.804,A -85,B 0,C 180,E1 23228.49,E2 23228.49} C_VEL
LIN {X 0,Y 230.101,Z 898.59,A -85,B 0,C 180,E1 23229.778,E2 23229.778} C_VEL
LIN {X 0,Y 185.761,Z 947.204,A -85,B 0,C 180,E1 23238.241,E2 23238.241} C_VEL
LIN {X 0,Y 141.67,Z 983.277,A -85,B 0,C 180,E1 23253.926,E2 23253.926} C_VEL
LIN {X 0,Y 112.094,Z 1005.073,A -85,B 0,C 180,E1 23281.711,E2 23281.711} C_VEL
LIN {X 0,Y 106.965,Z 1011.315,A -85,B 0,C 180,E1 23305.928,E2 23305.928} C_VEL
LIN {X 0,Y 108.961,Z 1010.559,A -85,B 0,C 180,E1 23330.373,E2 23330.373} C_VEL
LIN {X 0,Y 135.733,Z 997.804,A -85,B 0,C 180,E1 23362.158,E2 23362.158} C_VEL
LIN {X 0,Y 193,Z 967.642,A -85,B 0,C 180,E1 23382.085,E2 23382.085} C_VEL
LIN {X 0,Y 207.053,Z 958.906,A -85,B 0,C 180,E1 23385.19,E2 23385.19} C_VEL
LIN {X 0,Y 149.433,Z 988.36,A -85,B 0,C 180,E1 23401.369,E2 23401.369} C_VEL
LIN {X 0,Y 113.596,Z 1002.289,A -85,B 0,C 180,E1 23429.737,E2 23429.737} C_VEL
LIN {X 0,Y 104.828,Z 1003.7,A -85,B 0,C 180,E1 23459.56,E2 23459.56} C_VEL
LIN {X 0,Y 114.062,Z 996.267,A -85,B 0,C 180,E1 23487.654,E2 23487.654} C_VEL
LIN {X 0,Y 143.499,Z 975.526,A -85,B 0,C 180,E1 23513.368,E2 23513.368} C_VEL
LIN {X 0,Y 184.614,Z 942.622,A -85,B 0,C 180,E1 23528.064,E2 23528.064} C_VEL
LIN {X 0,Y 202.517,Z 922.303,A -85,B 0,C 180,E1 23534.864,E2 23534.864} C_VEL
LIN {X 0,Y 223.079,Z 899.214,A -85,B 0,C 180,E1 23538.47,E2 23538.47} C_VEL
LIN {X 0,Y 224.896,Z 884.408,A -85,B 0,C 180,E1 23550.904,E2 23550.904} C_VEL
LIN {X 0,Y 225.841,Z 879.303,A -85,B 0,C 180,E1 23562.357,E2 23562.357} C_VEL
LIN {X 0,Y 227.871,Z 881.632,A -85,B 0,C 180,E1 23574.224,E2 23574.224} C_VEL
LIN {X 0,Y 227.206,Z 896.397,A -85,B 0,C 180,E1 23586.372,E2 23586.372} C_VEL
LIN {X 0,Y 225.048,Z 901.35,A -85,B 0,C 180,E1 23588.201,E2 23588.201} C_VEL
LIN {X 0,Y 180.007,Z 948.779,A -85,B 0,C 180,E1 23596.496,E2 23596.496} C_VEL
LIN {X 0,Y 134.643,Z 984.165,A -85,B 0,C 180,E1 23612.285,E2 23612.285} C_VEL
LIN {X 0,Y 104.935,Z 1004.526,A -85,B 0,C 180,E1 23639.586,E2 23639.586} C_VEL
LIN {X 0,Y 98.967,Z 1010.935,A -85,B 0,C 180,E1 23665.599,E2 23665.599} C_VEL
LIN {X 0,Y 101.319,Z 1010.333,A -85,B 0,C 180,E1 23691.987,E2 23691.987} C_VEL
LIN {X 0,Y 130.797,Z 997.906,A -85,B 0,C 180,E1 23725.035,E2 23725.035} C_VEL
LIN {X 0,Y 190.105,Z 968.733,A -85,B 0,C 180,E1 23744.306,E2 23744.306} C_VEL
LIN {X 0,Y 193.15,Z 967.04,A -85,B 0,C 180,E1 23745.143,E2 23745.143} C_VEL
LIN {X 0,Y 134.86,Z 993.243,A -85,B 0,C 180,E1 23763.299,E2 23763.299} C_VEL
LIN {X 0,Y 102.067,Z 1003.873,A -85,B 0,C 180,E1 23795.144,E2 23795.144} C_VEL
LIN {X 0,Y 97.611,Z 1002.959,A -85,B 0,C 180,E1 23827.132,E2 23827.132} C_VEL
LIN {X 0,Y 109.911,Z 994.322,A -85,B 0,C 180,E1 23853.962,E2 23853.962} C_VEL
LIN {X 0,Y 145.717,Z 970.559,A -85,B 0,C 180,E1 23879.236,E2 23879.236} C_VEL
LIN {X 0,Y 192.287,Z 932.363,A -85,B 0,C 180,E1 23892.902,E2 23892.902} C_VEL
LIN {X 0,Y 202.517,Z 922.303,A -85,B 0,C 180,E1 23894.864,E2 23894.864} C_VEL
LIN {X 0,Y 213.226,Z 907.916,A -85,B 0,C 180,E1 23899.262,E2 23899.262} C_VEL
LIN {X 0,Y 217.626,Z 902.65,A -85,B 0,C 180,E1 23900.117,E2 23900.117} C_VEL
LIN {X 0,Y 219.764,Z 890.145,A -85,B 0,C 180,E1 23911.568,E2 23911.568} C_VEL
LIN {X 0,Y 221.355,Z 885.306,A -85,B 0,C 180,E1 23926.073,E2 23926.073} C_VEL
LIN {X 0,Y 222.531,Z 889.555,A -85,B 0,C 180,E1 23936.045,E2 23936.045} C_VEL
LIN {X 0,Y 221.432,Z 902.488,A -85,B 0,C 180,E1 23946.386,E2 23946.386} C_VEL
LIN {X 0,Y 174.391,Z 950.32,A -85,B 0,C 180,E1 23954.627,E2 23954.627} C_VEL
LIN {X 0,Y 127.85,Z 984.85,A -85,B 0,C 180,E1 23970.404,E2 23970.404} C_VEL
LIN {X 0,Y 96.591,Z 1004.861,A -85,B 0,C 180,E1 23999.553,E2 23999.553} C_VEL
LIN {X 0,Y 90.939,Z 1010.548,A -85,B 0,C 180,E1 24025.209,E2 24025.209} C_VEL
LIN {X 0,Y 93.759,Z 1010.112,A -85,B 0,C 180,E1 24053.865,E2 24053.865} C_VEL
LIN {X 0,Y 126.033,Z 998.093,A -85,B 0,C 180,E1 24088.046,E2 24088.046} C_VEL
LIN {X 0,Y 178.179,Z 974.77,A -85,B 0,C 180,E1 24105.258,E2 24105.258} C_VEL
LIN {X 0,Y 118.887,Z 997.807,A -85,B 0,C 180,E1 24126.645,E2 24126.645} C_VEL
LIN {X 0,Y 94.047,Z 1004.394,A -85,B 0,C 180,E1 24154.507,E2 24154.507} C_VEL
LIN {X 0,Y 89.846,Z 1003.008,A -85,B 0,C 180,E1 24188.549,E2 24188.549} C_VEL
LIN {X 0,Y 104.816,Z 993.418,A -85,B 0,C 180,E1 24218.329,E2 24218.329} C_VEL
LIN {X 0,Y 144.135,Z 968.579,A -85,B 0,C 180,E1 24242.991,E2 24242.991} C_VEL
LIN {X 0,Y 191.366,Z 930.495,A -85,B 0,C 180,E1 24255.542,E2 24255.542} C_VEL
LIN {X 0,Y 213.226,Z 907.916,A -85,B 0,C 180,E1 24259.262,E2 24259.262} C_VEL
LIN {X 0,Y 214.751,Z 903.581,A -85,B 0,C 180,E1 24261.871,E2 24261.871} C_VEL
LIN {X 0,Y 213.167,Z 901.805,A -85,B 0,C 180,E1 24265.502,E2 24265.502} C_VEL
LIN {X 0,Y 214.861,Z 893.217,A -85,B 0,C 180,E1 24277.096,E2 24277.096} C_VEL
LIN {X 0,Y 216.985,Z 892.016,A -85,B 0,C 180,E1 24289.886,E2 24289.886} C_VEL
LIN {X 0,Y 216.74,Z 899.951,A -85,B 0,C 180,E1 24300.164,E2 24300.164} C_VEL
LIN {X 0,Y 215.355,Z 906.718,A -85,B 0,C 180,E1 24304.856,E2 24304.856} C_VEL
LIN {X 0,Y 165.563,Z 954.648,A -85,B 0,C 180,E1 24313.395,E2 24313.395} C_VEL
LIN {X 0,Y 115.602,Z 988.988,A -85,B 0,C 180,E1 24331.421,E2 24331.421} C_VEL
LIN {X 0,Y 86.381,Z 1006.438,A -85,B 0,C 180,E1 24363.941,E2 24363.941} C_VEL
LIN {X 0,Y 82.995,Z 1010.81,A -85,B 0,C 180,E1 24395.241,E2 24395.241} C_VEL
LIN {X 0,Y 97.757,Z 1006.374,A -85,B 0,C 180,E1 24434.308,E2 24434.308} C_VEL
LIN {X 0,Y 151.639,Z 986.732,A -85,B 0,C 180,E1 24461.935,E2 24461.935} C_VEL
LIN {X 0,Y 163.327,Z 981.528,A -85,B 0,C 180,E1 24465.382,E2 24465.382} C_VEL
LIN {X 0,Y 104.951,Z 1000.941,A -85,B 0,C 180,E1 24489.763,E2 24489.763} C_VEL
LIN {X 0,Y 83.71,Z 1005.113,A -85,B 0,C 180,E1 24519.529,E2 24519.529} C_VEL
LIN {X 0,Y 85.05,Z 1001.222,A -85,B 0,C 180,E1 24559.489,E2 24559.489} C_VEL
LIN {X 0,Y 111.329,Z 986.213,A -85,B 0,C 180,E1 24592.02,E2 24592.02} C_VEL
LIN {X 0,Y 158.174,Z 955.902,A -85,B 0,C 180,E1 24611.274,E2 24611.274} C_VEL
LIN {X 0,Y 207.453,Z 911.714,A -85,B 0,C 180,E1 24620.85,E2 24620.85} C_VEL
LIN {X 0,Y 211.574,Z 907.134,A -85,B 0,C 180,E1 24621.447,E2 24621.447} C_VEL
LIN {X 0,Y 213.167,Z 901.805,A -85,B 0,C 180,E1 24625.502,E2 24625.502} C_VEL
LIN {X 0,Y 209.259,Z 900.061,A -85,B 0,C 180,E1 24635.163,E2 24635.163} C_VEL
LIN {X 0,Y 211.56,Z 897.927,A -85,B 0,C 180,E1 24649.623,E2 24649.623} C_VEL
LIN {X 0,Y 211.083,Z 905.842,A -85,B 0,C 180,E1 24660.053,E2 24660.053} C_VEL
LIN {X 0,Y 209.625,Z 910.425,A -85,B 0,C 180,E1 24663.215,E2 24663.215} C_VEL
LIN {X 0,Y 160.509,Z 955.767,A -85,B 0,C 180,E1 24671.191,E2 24671.191} C_VEL
LIN {X 0,Y 111.452,Z 988.076,A -85,B 0,C 180,E1 24687.731,E2 24687.731} C_VEL
LIN {X 0,Y 79.089,Z 1005.912,A -85,B 0,C 180,E1 24721.328,E2 24721.328} C_VEL
LIN {X 0,Y 74.961,Z 1010.474,A -85,B 0,C 180,E1 24755.804,E2 24755.804} C_VEL
LIN {X 0,Y 91.998,Z 1006.33,A -85,B 0,C 180,E1 24797.922,E2 24797.922} C_VEL
LIN {X 0,Y 148.971,Z 987.266,A -85,B 0,C 180,E1 24825.405,E2 24825.405} C_VEL
LIN {X 0,Y 99.285,Z 1001.633,A -85,B 0,C 180,E1 24846.554,E2 24846.554} C_VEL
LIN {X 0,Y 73.685,Z 1005.403,A -85,B 0,C 180,E1 24886.307,E2 24886.307} C_VEL
LIN {X 0,Y 81.318,Z 999.329,A -85,B 0,C 180,E1 24929.546,E2 24929.546} C_VEL
LIN {X 0,Y 115.961,Z 980.791,A -85,B 0,C 180,E1 24960.869,E2 24960.869} C_VEL
LIN {X 0,Y 165.824,Z 947.691,A -85,B 0,C 180,E1 24976.436,E2 24976.436} C_VEL
LIN {X 0,Y 206.615,Z 910.328,A -85,B 0,C 180,E1 24983.207,E2 24983.207} C_VEL
LIN {X 0,Y 209.259,Z 900.061,A -85,B 0,C 180,E1 24995.163,E2 24995.163} C_VEL
LIN {X 0,Y 205.223,Z 903.514,A -85,B 0,C 180,E1 25004.92,E2 25004.92} C_VEL
LIN {X 0,Y 206.069,Z 907.31,A -85,B 0,C 180,E1 25015.729,E2 25015.729} C_VEL
LIN {X 0,Y 204.031,Z 914.112,A -85,B 0,C 180,E1 25021.473,E2 25021.473} C_VEL
LIN {X 0,Y 153.077,Z 958.775,A -85,B 0,C 180,E1 25029.398,E2 25029.398} C_VEL
LIN {X 0,Y 102.515,Z 989.932,A -85,B 0,C 180,E1 25046.485,E2 25046.485} C_VEL
LIN {X 0,Y 69.786,Z 1006.626,A -85,B 0,C 180,E1 25084.213,E2 25084.213} C_VEL
LIN {X 0,Y 66.951,Z 1010.138,A -85,B 0,C 180,E1 25116.502,E2 25116.502} C_VEL
LIN {X 0,Y 87.573,Z 1006.05,A -85,B 0,C 180,E1 25162.816,E2 25162.816} C_VEL
LIN {X 0,Y 134.611,Z 992.245,A -85,B 0,C 180,E1 25185.449,E2 25185.449} C_VEL
LIN {X 0,Y 79.225,Z 1004.905,A -85,B 0,C 180,E1 25216.827,E2 25216.827} C_VEL
LIN {X 0,Y 64.567,Z 1005.161,A -85,B 0,C 180,E1 25255.604,E2 25255.604} C_VEL
LIN {X 0,Y 76.273,Z 998.421,A -85,B 0,C 180,E1 25295.715,E2 25295.715} C_VEL
LIN {X 0,Y 115.868,Z 978.602,A -85,B 0,C 180,E1 25326.118,E2 25326.118} C_VEL
LIN {X 0,Y 168.27,Z 943.686,A -85,B 0,C 180,E1 25340.053,E2 25340.053} C_VEL
LIN {X 0,Y 201.368,Z 913.355,A -85,B 0,C 180,E1 25345.531,E2 25345.531} C_VEL
LIN {X 0,Y 203.762,Z 905.61,A -85,B 0,C 180,E1 25355.771,E2 25355.771} C_VEL
LIN {X 0,Y 205.223,Z 903.514,A -85,B 0,C 180,E1 25364.92,E2 25364.92} C_VEL
LIN {X 0,Y 201.638,Z 909.609,A -85,B 0,C 180,E1 25372.15,E2 25372.15} C_VEL
LIN {X 0,Y 200.457,Z 912.183,A -85,B 0,C 180,E1 25374.633,E2 25374.633} C_VEL
LIN {X 0,Y 198.318,Z 917.847,A -85,B 0,C 180,E1 25379.679,E2 25379.679} C_VEL
LIN {X 0,Y 145.412,Z 961.98,A -85,B 0,C 180,E1 25387.469,E2 25387.469} C_VEL
LIN {X 0,Y 92.523,Z 992.16,A -85,B 0,C 180,E1 25405.551,E2 25405.551} C_VEL
LIN {X 0,Y 60.602,Z 1007.287,A -85,B 0,C 180,E1 25447.93,E2 25447.93} C_VEL
LIN {X 0,Y 58.926,Z 1009.797,A -85,B 0,C 180,E1 25477.392,E2 25477.392} C_VEL
LIN {X 0,Y 81.804,Z 1006.185,A -85,B 0,C 180,E1 25526.588,E2 25526.588} C_VEL
LIN {X 0,Y 119.367,Z 996.715,A -85,B 0,C 180,E1 25545.696,E2 25545.696} C_VEL
LIN {X 0,Y 67.624,Z 1005.865,A -85,B 0,C 180,E1 25579.824,E2 25579.824} C_VEL
LIN {X 0,Y 57.282,Z 1004.26,A -85,B 0,C 180,E1 25628.451,E2 25628.451} C_VEL
LIN {X 0,Y 78.687,Z 994.607,A -85,B 0,C 180,E1 25669.999,E2 25669.999} C_VEL
LIN {X 0,Y 127.535,Z 970.003,A -85,B 0,C 180,E1 25694.555,E2 25694.555} C_VEL
LIN {X 0,Y 180.909,Z 931.52,A -85,B 0,C 180,E1 25704.879,E2 25704.879} C_VEL
LIN {X 0,Y 195.843,Z 917.328,A -85,B 0,C 180,E1 25707.144,E2 25707.144} C_VEL
LIN {X 0,Y 198.635,Z 910.059,A -85,B 0,C 180,E1 25719.842,E2 25719.842} C_VEL
LIN {X 0,Y 200.417,Z 909.47,A -85,B 0,C 180,E1 25729.039,E2 25729.039} C_VEL
LIN {X 0,Y 200.457,Z 912.183,A -85,B 0,C 180,E1 25734.633,E2 25734.633} C_VEL
LIN {X 0,Y 193.557,Z 920.618,A -85,B 0,C 180,E1 25737.513,E2 25737.513} C_VEL
LIN {X 0,Y 186.74,Z 927.187,A -85,B 0,C 180,E1 25738.408,E2 25738.408} C_VEL
LIN {X 0,Y 132.266,Z 968.487,A -85,B 0,C 180,E1 25746.502,E2 25746.502} C_VEL
LIN {X 0,Y 77.282,Z 996.428,A -85,B 0,C 180,E1 25767.901,E2 25767.901} C_VEL
LIN {X 0,Y 53.165,Z 1006.758,A -85,B 0,C 180,E1 25804.64,E2 25804.64} C_VEL
LIN {X 0,Y 50.923,Z 1009.433,A -85,B 0,C 180,E1 25838.562,E2 25838.562} C_VEL
LIN {X 0,Y 77.541,Z 1006.096,A -85,B 0,C 180,E1 25891.718,E2 25891.718} C_VEL
LIN {X 0,Y 103.992,Z 1000.438,A -85,B 0,C 180,E1 25905.863,E2 25905.863} C_VEL
LIN {X 0,Y 55.894,Z 1006.461,A -85,B 0,C 180,E1 25944.224,E2 25944.224} C_VEL
LIN {X 0,Y 53.472,Z 1002.553,A -85,B 0,C 180,E1 26005.122,E2 26005.122} C_VEL
LIN {X 0,Y 87.477,Z 988.798,A -85,B 0,C 180,E1 26044.326,E2 26044.326} C_VEL
LIN {X 0,Y 144.15,Z 958.102,A -85,B 0,C 180,E1 26062.152,E2 26062.152} C_VEL
LIN {X 0,Y 190.31,Z 921.464,A -85,B 0,C 180,E1 26068.726,E2 26068.726} C_VEL
LIN {X 0,Y 192.69,Z 915.914,A -85,B 0,C 180,E1 26079.192,E2 26079.192} C_VEL
LIN {X 0,Y 194.647,Z 915.115,A -85,B 0,C 180,E1 26088.71,E2 26088.71} C_VEL
LIN {X 0,Y 193.614,Z 920.629,A -85,B 0,C 180,E1 26097.702,E2 26097.702} C_VEL
LIN {X 0,Y 186.74,Z 927.187,A -85,B 0,C 180,E1 26098.408,E2 26098.408} C_VEL
LIN {X 0,Y 158.641,Z 948.849,A -85,B 0,C 180,E1 26098.826,E2 26098.826} C_VEL
LIN {X 0,Y 102.612,Z 982.964,A -85,B 0,C 180,E1 26109.573,E2 26109.573} C_VEL
LIN {X 0,Y 52.693,Z 1003.51,A -85,B 0,C 180,E1 26143.934,E2 26143.934} C_VEL
LIN {X 0,Y 42.927,Z 1008.023,A -85,B 0,C 180,E1 26179.809,E2 26179.809} C_VEL
LIN {X 0,Y 49.475,Z 1008.98,A -85,B 0,C 180,E1 26230.261,E2 26230.261} C_VEL
LIN {X 0,Y 89.983,Z 1003.196,A -85,B 0,C 180,E1 26265.465,E2 26265.465} C_VEL
LIN {X 0,Y 44.132,Z 1006.633,A -85,B 0,C 180,E1 26311.31,E2 26311.31} C_VEL
LIN {X 0,Y 50.603,Z 1001.129,A -85,B 0,C 180,E1 26378.632,E2 26378.632} C_VEL
LIN {X 0,Y 95.421,Z 983.667,A -85,B 0,C 180,E1 26414.164,E2 26414.164} C_VEL
LIN {X 0,Y 153.763,Z 950.252,A -85,B 0,C 180,E1 26427.032,E2 26427.032} C_VEL
LIN {X 0,Y 184.791,Z 925.277,A -85,B 0,C 180,E1 26430.779,E2 26430.779} C_VEL
LIN {X 0,Y 187.644,Z 920.594,A -85,B 0,C 180,E1 26443.505,E2 26443.505} C_VEL
LIN {X 0,Y 188.968,Z 922.107,A -85,B 0,C 180,E1 26453.029,E2 26453.029} C_VEL
LIN {X 0,Y 187.125,Z 925.279,A -85,B 0,C 180,E1 26455.807,E2 26455.807} C_VEL
LIN {X 0,Y 158.641,Z 948.849,A -85,B 0,C 180,E1 26458.826,E2 26458.826} C_VEL
LIN {X 0,Y 128.436,Z 967.511,A -85,B 0,C 180,E1 26459.573,E2 26459.573} C_VEL
LIN {X 0,Y 71.021,Z 994.719,A -85,B 0,C 180,E1 26475.916,E2 26475.916} C_VEL
LIN {X 0,Y 39.044,Z 1005.591,A -85,B 0,C 180,E1 26514.323,E2 26514.323} C_VEL
LIN {X 0,Y 35.013,Z 1008.58,A -85,B 0,C 180,E1 26562.505,E2 26562.505} C_VEL
LIN {X 0,Y 71.174,Z 1005.954,A -85,B 0,C 180,E1 26623.617,E2 26623.617} C_VEL
LIN {X 0,Y 73.027,Z 1005.613,A -85,B 0,C 180,E1 26626.244,E2 26626.244} C_VEL
LIN {X 0,Y 32.943,Z 1006.289,A -85,B 0,C 180,E1 26684.121,E2 26684.121} C_VEL
LIN {X 0,Y 47.317,Z 1000.28,A -85,B 0,C 180,E1 26749.307,E2 26749.307} C_VEL
LIN {X 0,Y 98.383,Z 981.101,A -85,B 0,C 180,E1 26780.474,E2 26780.474} C_VEL
LIN {X 0,Y 155.479,Z 947.963,A -85,B 0,C 180,E1 26790.364,E2 26790.364} C_VEL
LIN {X 0,Y 179.232,Z 929.257,A -85,B 0,C 180,E1 26792.76,E2 26792.76} C_VEL
LIN {X 0,Y 182.609,Z 925.913,A -85,B 0,C 180,E1 26807.955,E2 26807.955} C_VEL
LIN {X 0,Y 181.746,Z 928.704,A -85,B 0,C 180,E1 26813.692,E2 26813.692} C_VEL
LIN {X 0,Y 128.436,Z 967.511,A -85,B 0,C 180,E1 26819.573,E2 26819.573} C_VEL
LIN {X 0,Y 96.524,Z 982.814,A -85,B 0,C 180,E1 26821.059,E2 26821.059} C_VEL
LIN {X 0,Y 38.543,Z 1003.425,A -85,B 0,C 180,E1 26853.993,E2 26853.993} C_VEL
LIN {X 0,Y 27.156,Z 1008.147,A -85,B 0,C 180,E1 26926.21,E2 26926.21} C_VEL
LIN {X 0,Y 58.798,Z 1007.017,A -85,B 0,C 180,E1 26985.567,E2 26985.567} C_VEL
LIN {X 0,Y 26.564,Z 1006.775,A -85,B 0,C 180,E1 27031.054,E2 27031.054} C_VEL
LIN {X 0,Y 43.465,Z 999.958,A -85,B 0,C 180,E1 27118.752,E2 27118.752} C_VEL
LIN {X 0,Y 100.69,Z 979.23,A -85,B 0,C 180,E1 27145.999,E2 27145.999} C_VEL
LIN {X 0,Y 160.567,Z 943.555,A -85,B 0,C 180,E1 27153.888,E2 27153.888} C_VEL
LIN {X 0,Y 173.593,Z 933.342,A -85,B 0,C 180,E1 27155.184,E2 27155.184} C_VEL
LIN {X 0,Y 176.455,Z 931.483,A -85,B 0,C 180,E1 27169.28,E2 27169.28} C_VEL
LIN {X 0,Y 175.285,Z 933.221,A -85,B 0,C 180,E1 27171.535,E2 27171.535} C_VEL
LIN {X 0,Y 116.436,Z 972.975,A -85,B 0,C 180,E1 27177.455,E2 27177.455} C_VEL
LIN {X 0,Y 96.524,Z 982.814,A -85,B 0,C 180,E1 27181.059,E2 27181.059} C_VEL
LIN {X 0,Y 63.163,Z 994.61,A -85,B 0,C 180,E1 27183.987,E2 27183.987} C_VEL
LIN {X 0,Y 19.52,Z 1006.476,A -85,B 0,C 180,E1 27247.103,E2 27247.103} C_VEL
LIN {X 0,Y 27.363,Z 1008.142,A -85,B 0,C 180,E1 27326.269,E2 27326.269} C_VEL
LIN {X 0,Y 41.181,Z 1007.833,A -85,B 0,C 180,E1 27346.017,E2 27346.017} C_VEL
LIN {X 0,Y 24.434,Z 1003.466,A -85,B 0,C 180,E1 27468.11,E2 27468.11} C_VEL
LIN {X 0,Y 70.285,Z 990.884,A -85,B 0,C 180,E1 27504.077,E2 27504.077} C_VEL
LIN {X 0,Y 132.444,Z 961.825,A -85,B 0,C 180,E1 27514.475,E2 27514.475} C_VEL
LIN {X 0,Y 167.226,Z 937.959,A -85,B 0,C 180,E1 27517.251,E2 27517.251} C_VEL
LIN {X 0,Y 170.221,Z 936.472,A -85,B 0,C 180,E1 27529.032,E2 27529.032} C_VEL
LIN {X 0,Y 110.66,Z 975.025,A -85,B 0,C 180,E1 27534.079,E2 27534.079} C_VEL
LIN {X 0,Y 63.163,Z 994.61,A -85,B 0,C 180,E1 27543.987,E2 27543.987} C_VEL
LIN {X 0,Y 29.005,Z 1002.691,A -85,B 0,C 180,E1 27551.784,E2 27551.784} C_VEL
LIN {X 0,Y 12.429,Z 1007.259,A -85,B 0,C 180,E1 27667.585,E2 27667.585} C_VEL
LIN {X 0,Y 23.624,Z 1007.758,A -85,B 0,C 180,E1 27704.426,E2 27704.426} C_VEL
LIN {X 0,Y 31.37,Z 1001.251,A -85,B 0,C 180,E1 27856.542,E2 27856.542} C_VEL
LIN {X 0,Y 92.499,Z 981.86,A -85,B 0,C 180,E1 27874.48,E2 27874.48} C_VEL
LIN {X 0,Y 152.174,Z 948.868,A -85,B 0,C 180,E1 27879.225,E2 27879.225} C_VEL
LIN {X 0,Y 160.917,Z 942.653,A -85,B 0,C 180,E1 27879.709,E2 27879.709} C_VEL
LIN {X 0,Y 163.435,Z 941.163,A -85,B 0,C 180,E1 27886.517,E2 27886.517} C_VEL
LIN {X 0,Y 103.886,Z 977.498,A -85,B 0,C 180,E1 27890.444,E2 27890.444} C_VEL
LIN {X 0,Y 45.05,Z 998.945,A -85,B 0,C 180,E1 27901.891,E2 27901.891} C_VEL
LIN {X 0,Y 29.005,Z 1002.691,A -85,B 0,C 180,E1 27911.784,E2 27911.784} C_VEL
LIN {X 0,Y 5.278,Z 1005.678,A -85,B 0,C 180,E1 27921.156,E2 27921.156} C_VEL
LIN {X 0,Y 0.418,Z 1006.098,A -85,B 0,C 180,E1 28045.457,E2 28045.457} C_VEL
LIN {X 0,Y 42.298,Z 998.506,A -85,B 0,C 180,E1 27873.783,E2 27873.783} C_VEL
LIN {X 0,Y 107.616,Z 974.932,A -85,B 0,C 180,E1 27880.341,E2 27880.341} C_VEL
LIN {X 0,Y 155.352,Z 946.621,A -85,B 0,C 180,E1 27882.363,E2 27882.363} C_VEL
LIN {X 0,Y 156.144,Z 946.174,A -85,B 0,C 180,E1 27883.882,E2 27883.882} C_VEL
LIN {X 0,Y 94.369,Z 981.34,A -85,B 0,C 180,E1 27886.557,E2 27886.557} C_VEL
LIN {X 0,Y 30.486,Z 1001.572,A -85,B 0,C 180,E1 27894.76,E2 27894.76} C_VEL
LIN {X 0,Y 5.278,Z 1005.678,A -85,B 0,C 180,E1 27921.156,E2 27921.156} C_VEL
LIN {X 0,Y 3.435,Z 1007.672,A -85,B 0,C 180,E1 27923.084,E2 27923.084} C_VEL
LIN {X 0,Y 3.435,Z 1028,A -85,B 0,C 180,E1 27923.084,E2 27923.084} C_VEL
LIN {X 0,Y 3.435,Z 1028,A -85,B 0,C 180,E1 27923.084,E2 27923.084}

QRS_NEXT_CUT()
PTP {E1 27896.865,E2 27896.865}
PTP {X 0,Y 607.915,A -85,B 0,C 180,E1 27896.865,E2 27896.865,E3 0,E4 0,E5 0,E6 0}
QRS_SPEED_INIT()
LIN {X 0,Y 607.915,Z 1028,A -85,B 0,C 180,E1 27896.865,E2 27896.865,E3 0,E4 0,E5 0,E6 0} C_VEL
LIN {X 0,Y 607.915,Z 365.399,A -85,B 0,C 180,E1 27896.865,E2 27896.865} C_VEL
LIN {X 0,Y 607.915,Z 357.322,A -85,B 0,C 180,E1 27896.865,E2 27896.865} C_VEL
LIN {X 0,Y 607.888,Z 355.322,A -85,B 0,C 180,E1 27896.676,E2 27896.676} C_VEL
LIN {X 0,Y 607.853,Z 355.325,A -85,B 0,C 180,E1 27893.767,E2 27893.767} C_VEL
LIN {X 0,Y 607.909,Z 355.321,A -85,B 0,C 180,E1 27890.628,E2 27890.628} C_VEL
LIN {X 0,Y 607.855,Z 355.324,A -85,B 0,C 180,E1 27887.652,E2 27887.652} C_VEL
LIN {X 0,Y 607.919,Z 355.32,A -85,B 0,C 180,E1 27884.521,E2 27884.521} C_VEL
LIN {X 0,Y 607.859,Z 355.324,A -85,B 0,C 180,E1 27881.49,E2 27881.49} C_VEL
LIN {X 0,Y 607.912,Z 355.32,A -85,B 0,C 180,E1 27878.311,E2 27878.311} C_VEL
LIN {X 0,Y 607.863,Z 355.324,A -85,B 0,C 180,E1 27875.304,E2 27875.304} C_VEL
LIN {X 0,Y 607.917,Z 355.32,A -85,B 0,C 180,E1 27872.153,E2 27872.153} C_VEL
LIN {X 0,Y 607.868,Z 355.323,A -85,B 0,C 180,E1 27869.123,E2 27869.123} C_VEL
LIN {X 0,Y 607.915,Z 355.32,A -85,B 0,C 180,E1 27865.983,E2 27865.983} C_VEL
LIN {X 0,Y 607.873,Z 355.324,A -85,B 0,C 180,E1 27862.867,E2 27862.867} C_VEL
LIN {X 0,Y 607.914,Z 355.317,A -85,B 0,C 180,E1 27859.607,E2 27859.607} C_VEL
LIN {X 0,Y 607.901,Z 355.326,A -85,B 0,C 180,E1 27856.355,E2 27856.355} C_VEL
LIN {X 0,Y 607.885,Z 355.319,A -85,B 0,C 180,E1 27853.088,E2 27853.088} C_VEL
LIN {X 0,Y 607.915,Z 355.326,A -85,B 0,C 180,E1 27849.964,E2 27849.964} C_VEL
LIN {X 0,Y 607.884,Z 355.32,A -85,B 0,C 180,E1 27846.771,E2 27846.771} C_VEL
LIN {X 0,Y 607.908,Z 355.324,A -85,B 0,C 180,E1 27843.657,E2 27843.657} C_VEL
LIN {X 0,Y 607.884,Z 355.32,A -85,B 0,C 180,E1 27840.471,E2 27840.471} C_VEL
LIN {X 0,Y 607.903,Z 355.321,A -85,B 0,C 180,E1 27837.312,E2 27837.312} C_VEL
LIN {X 0,Y 607.888,Z 355.322,A -85,B 0,C 180,E1 27834.173,E2 27834.173} C_VEL
LIN {X 0,Y 607.901,Z 355.32,A -85,B 0,C 180,E1 27831.008,E2 27831.008} C_VEL
LIN {X 0,Y 607.893,Z 355.323,A -85,B 0,C 180,E1 27827.91,E2 27827.91} C_VEL
LIN {X 0,Y 607.903,Z 355.318,A -85,B 0,C 180,E1 27824.732,E2 27824.732} C_VEL
LIN {X 0,Y 607.909,Z 355.325,A -85,B 0,C 180,E1 27821.476,E2 27821.476} C_VEL
LIN {X 0,Y 607.908,Z 355.313,A -85,B 0,C 180,E1 27818.129,E2 27818.129} C_VEL
LIN {X 0,Y 607.897,Z 355.344,A -85,B 0,C 180,E1 27815.756,E2 27815.756} C_VEL
LIN {X 0,Y 607.91,Z 361.597,A -85,B 0,C 180,E1 27815.318,E2 27815.318} C_VEL
LIN {X 0,Y 607.919,Z 559.44,A -85,B 0,C 180,E1 27812.484,E2 27812.484} C_VEL
LIN {X 0,Y 607.913,Z 709.494,A -85,B 0,C 180,E1 27810.374,E2 27810.374} C_VEL
LIN {X 0,Y 607.915,Z 732.303,A -85,B 0,C 180,E1 27809.88,E2 27809.88} C_VEL
LIN {X 0,Y 607.914,Z 751.657,A -85,B 0,C 180,E1 27809.314,E2 27809.314} C_VEL
LIN {X 0,Y 607.91,Z 773.027,A -85,B 0,C 180,E1 27808.537,E2 27808.537} C_VEL
LIN {X 0,Y 607.919,Z 792.942,A -85,B 0,C 180,E1 27807.641,E2 27807.641} C_VEL
LIN {X 0,Y 607.915,Z 813.593,A -85,B 0,C 180,E1 27806.556,E2 27806.556} C_VEL
LIN {X 0,Y 607.917,Z 832.95,A -85,B 0,C 180,E1 27805.35,E2 27805.35} C_VEL
LIN {X 0,Y 607.915,Z 852.582,A -85,B 0,C 180,E1 27803.955,E2 27803.955} C_VEL
LIN {X 0,Y 607.906,Z 871.08,A -85,B 0,C 180,E1 27802.437,E2 27802.437} C_VEL
LIN {X 0,Y 607.903,Z 889.328,A -85,B 0,C 180,E1 27800.722,E2 27800.722} C_VEL
LIN {X 0,Y 607.903,Z 905.458,A -85,B 0,C 180,E1 27798.999,E2 27798.999} C_VEL
LIN {X 0,Y 607.904,Z 920.372,A -85,B 0,C 180,E1 27797.169,E2 27797.169} C_VEL
LIN {X 0,Y 607.91,Z 934.177,A -85,B 0,C 180,E1 27795.228,E2 27795.228} C_VEL
LIN {X 0,Y 607.917,Z 946.274,A -85,B 0,C 180,E1 27793.27,E2 27793.27} C_VEL
LIN {X 0,Y 607.915,Z 956.641,A -85,B 0,C 180,E1 27791.291,E2 27791.291} C_VEL
LIN {X 0,Y 607.916,Z 965.583,A -85,B 0,C 180,E1 27789.289,E2 27789.289} C_VEL
LIN {X 0,Y 607.916,Z 973.269,A -85,B 0,C 180,E1 27787.158,E2 27787.158} C_VEL
LIN {X 0,Y 607.914,Z 979.204,A -85,B 0,C 180,E1 27785.097,E2 27785.097} C_VEL
LIN {X 0,Y 607.898,Z 983.743,A -85,B 0,C 180,E1 27782.894,E2 27782.894} C_VEL
LIN {X 0,Y 607.913,Z 986.658,A -85,B 0,C 180,E1 27780.757,E2 27780.757} C_VEL
LIN {X 0,Y 607.898,Z 987.851,A -85,B 0,C 180,E1 27778.61,E2 27778.61} C_VEL
LIN {X 0,Y 607.901,Z 987.631,A -85,B 0,C 180,E1 27776.502,E2 27776.502} C_VEL
LIN {X 0,Y 607.908,Z 985.887,A -85,B 0,C 180,E1 27774.504,E2 27774.504} C_VEL
LIN {X 0,Y 607.89,Z 982.694,A -85,B 0,C 180,E1 27772.393,E2 27772.393} C_VEL
LIN {X 0,Y 607.916,Z 977.909,A -85,B 0,C 180,E1 27770.33,E2 27770.33} C_VEL
LIN {X 0,Y 607.899,Z 971.602,A -85,B 0,C 180,E1 27768.229,E2 27768.229} C_VEL
LIN {X 0,Y 607.897,Z 963.685,A -85,B 0,C 180,E1 27766.174,E2 27766.174} C_VEL
LIN {X 0,Y 607.915,Z 954.554,A -85,B 0,C 180,E1 27764.183,E2 27764.183} C_VEL
LIN {X 0,Y 607.911,Z 943.994,A -85,B 0,C 180,E1 27762.256,E2 27762.256} C_VEL
LIN {X 0,Y 607.915,Z 931.482,A -85,B 0,C 180,E1 27760.27,E2 27760.27} C_VEL
LIN {X 0,Y 607.916,Z 917.565,A -85,B 0,C 180,E1 27758.381,E2 27758.381} C_VEL
LIN {X 0,Y 607.916,Z 901.382,A -85,B 0,C 180,E1 27756.458,E2 27756.458} C_VEL
LIN {X 0,Y 607.912,Z 884.924,A -85,B 0,C 180,E1 27754.744,E2 27754.744} C_VEL
LIN {X 0,Y 607.912,Z 866.696,A -85,B 0,C 180,E1 27753.097,E2 27753.097} C_VEL
LIN {X 0,Y 607.911,Z 846.941,A -85,B 0,C 180,E1 27751.536,E2 27751.536} C_VEL
LIN {X 0,Y 607.914,Z 827.795,A -85,B 0,C 180,E1 27750.218,E2 27750.218} C_VEL
LIN {X 0,Y 607.919,Z 807.588,A -85,B 0,C 180,E1 27749.025,E2 27749.025} C_VEL
LIN {X 0,Y 607.918,Z 787.67,A -85,B 0,C 180,E1 27748.013,E2 27748.013} C_VEL
LIN {X 0,Y 607.915,Z 766.01,A -85,B 0,C 180,E1 27747.103,E2 27747.103} C_VEL
LIN {X 0,Y 607.915,Z 746.09,A -85,B 0,C 180,E1 27746.417,E2 27746.417} C_VEL
LIN {X 0,Y 607.918,Z 723.272,A -85,B 0,C 180,E1 27745.814,E2 27745.814} C_VEL
LIN {X 0,Y 607.916,Z 704.178,A -85,B 0,C 180,E1 27745.449,E2 27745.449} C_VEL
LIN {X 0,Y 607.918,Z 479.215,A -85,B 0,C 180,E1 27742.292,E2 27742.292} C_VEL
LIN {X 0,Y 607.918,Z 361.342,A -85,B 0,C 180,E1 27740.583,E2 27740.583} C_VEL
LIN {X 0,Y 607.909,Z 355.608,A -85,B 0,C 180,E1 27740.144,E2 27740.144} C_VEL
LIN {X 0,Y 607.894,Z 355.321,A -85,B 0,C 180,E1 27738.608,E2 27738.608} C_VEL
LIN {X 0,Y 607.897,Z 355.316,A -85,B 0,C 180,E1 27735.258,E2 27735.258} C_VEL
LIN {X 0,Y 607.907,Z 355.324,A -85,B 0,C 180,E1 27732.057,E2 27732.057} C_VEL
LIN {X 0,Y 607.894,Z 355.32,A -85,B 0,C 180,E1 27728.894,E2 27728.894} C_VEL
LIN {X 0,Y 607.896,Z 355.323,A -85,B 0,C 180,E1 27725.759,E2 27725.759} C_VEL
LIN {X 0,Y 607.899,Z 355.322,A -85,B 0,C 180,E1 27722.64,E2 27722.64} C_VEL
LIN {X 0,Y 607.889,Z 355.322,A -85,B 0,C 180,E1 27719.529,E2 27719.529} C_VEL
LIN {X 0,Y 607.905,Z 355.323,A -85,B 0,C 180,E1 27716.417,E2 27716.417} C_VEL
LIN {X 0,Y 607.882,Z 355.321,A -85,B 0,C 180,E1 27713.294,E2 27713.294} C_VEL
LIN {X 0,Y 607.911,Z 355.326,A -85,B 0,C 180,E1 27710.134,E2 27710.134} C_VEL
LIN {X 0,Y 607.876,Z 355.321,A -85,B 0,C 180,E1 27707.074,E2 27707.074} C_VEL
LIN {X 0,Y 607.909,Z 355.327,A -85,B 0,C 180,E1 27703.851,E2 27703.851} C_VEL
LIN {X 0,Y 607.876,Z 355.321,A -85,B 0,C 180,E1 27700.76,E2 27700.76} C_VEL
LIN {X 0,Y 607.873,Z 355.326,A -85,B 0,C 180,E1 27697.465,E2 27697.465} C_VEL
LIN {X 0,Y 607.877,Z 355.322,A -85,B 0,C 180,E1 27694.473,E2 27694.473} C_VEL
LIN {X 0,Y 607.857,Z 355.326,A -85,B 0,C 180,E1 27691.251,E2 27691.251} C_VEL
LIN {X 0,Y 607.857,Z 355.325,A -85,B 0,C 180,E1 27688.437,E2 27688.437} C_VEL
LIN {X 0,Y 607.849,Z 355.327,A -85,B 0,C 180,E1 27685.167,E2 27685.167} C_VEL
LIN {X 0,Y 607.845,Z 355.327,A -85,B 0,C 180,E1 27682.3,E2 27682.3} C_VEL
LIN {X 0,Y 607.836,Z 355.328,A -85,B 0,C 180,E1 27678.98,E2 27678.98} C_VEL
LIN {X 0,Y 607.852,Z 355.328,A -85,B 0,C 180,E1 27676.095,E2 27676.095} C_VEL
LIN {X 0,Y 607.852,Z 355.324,A -85,B 0,C 180,E1 27672.923,E2 27672.923} C_VEL
LIN {X 0,Y 607.848,Z 355.316,A -85,B 0,C 180,E1 27670.153,E2 27670.153} C_VEL
LIN {X 0,Y 607.88,Z 355.635,A -85,B 0,C 180,E1 27669.781,E2 27669.781} C_VEL
LIN {X 0,Y 607.919,Z 363.193,A -85,B 0,C 180,E1 27669.226,E2 27669.226} C_VEL
LIN {X 0,Y 607.917,Z 391.172,A -85,B 0,C 180,E1 27667.368,E2 27667.368} C_VEL
LIN {X 0,Y 607.918,Z 591.55,A -85,B 0,C 180,E1 27664.499,E2 27664.499} C_VEL
LIN {X 0,Y 607.913,Z 739.031,A -85,B 0,C 180,E1 27662.426,E2 27662.426} C_VEL
LIN {X 0,Y 607.915,Z 761.996,A -85,B 0,C 180,E1 27661.932,E2 27661.932} C_VEL
LIN {X 0,Y 607.917,Z 780.551,A -85,B 0,C 180,E1 27661.394,E2 27661.394} C_VEL
LIN {X 0,Y 607.912,Z 801.888,A -85,B 0,C 180,E1 27660.629,E2 27660.629} C_VEL
LIN {X 0,Y 607.919,Z 822.107,A -85,B 0,C 180,E1 27659.726,E2 27659.726} C_VEL
LIN {X 0,Y 607.916,Z 842.732,A -85,B 0,C 180,E1 27658.65,E2 27658.65} C_VEL
LIN {X 0,Y 607.917,Z 862.537,A -85,B 0,C 180,E1 27657.423,E2 27657.423} C_VEL
LIN {X 0,Y 607.912,Z 881.936,A -85,B 0,C 180,E1 27656.051,E2 27656.051} C_VEL
LIN {X 0,Y 607.91,Z 900.181,A -85,B 0,C 180,E1 27654.558,E2 27654.558} C_VEL
LIN {X 0,Y 607.916,Z 918.579,A -85,B 0,C 180,E1 27652.842,E2 27652.842} C_VEL
LIN {X 0,Y 607.912,Z 934.86,A -85,B 0,C 180,E1 27651.114,E2 27651.114} C_VEL
LIN {X 0,Y 607.91,Z 950.073,A -85,B 0,C 180,E1 27649.252,E2 27649.252} C_VEL
LIN {X 0,Y 607.911,Z 964.504,A -85,B 0,C 180,E1 27647.223,E2 27647.223} C_VEL
LIN {X 0,Y 607.9,Z 976.023,A -85,B 0,C 180,E1 27645.358,E2 27645.358} C_VEL
LIN {X 0,Y 607.885,Z 986.744,A -85,B 0,C 180,E1 27643.315,E2 27643.315} C_VEL
LIN {X 0,Y 607.907,Z 995.299,A -85,B 0,C 180,E1 27641.401,E2 27641.401} C_VEL
LIN {X 0,Y 607.896,Z 1003.03,A -85,B 0,C 180,E1 27639.278,E2 27639.278} C_VEL
LIN {X 0,Y 607.888,Z 1008.584,A -85,B 0,C 180,E1 27637.373,E2 27637.373} C_VEL
LIN {X 0,Y 607.911,Z 1013.316,A -85,B 0,C 180,E1 27635.192,E2 27635.192} C_VEL
LIN {X 0,Y 607.882,Z 1016.063,A -85,B 0,C 180,E1 27633.303,E2 27633.303} C_VEL
LIN {X 0,Y 607.905,Z 1017.738,A -85,B 0,C 180,E1 27631.133,E2 27631.133} C_VEL
LIN {X 0,Y 607.886,Z 1017.806,A -85,B 0,C 180,E1 27629.154,E2 27629.154} C_VEL
LIN {X 0,Y 607.884,Z 1016.408,A -85,B 0,C 180,E1 27626.985,E2 27626.985} C_VEL
LIN {X 0,Y 607.907,Z 1013.643,A -85,B 0,C 180,E1 27625.002,E2 27625.002} C_VEL
LIN {X 0,Y 607.882,Z 1009.107,A -85,B 0,C 180,E1 27622.822,E2 27622.822} C_VEL
LIN {X 0,Y 607.904,Z 1003.351,A -85,B 0,C 180,E1 27620.823,E2 27620.823} C_VEL
LIN {X 0,Y 607.898,Z 995.796,A -85,B 0,C 180,E1 27618.716,E2 27618.716} C_VEL
LIN {X 0,Y 607.889,Z 987.233,A -85,B 0,C 180,E1 27616.787,E2 27616.787} C_VEL
LIN {X 0,Y 607.911,Z 977.198,A -85,B 0,C 180,E1 27614.843,E2 27614.843} C_VEL
LIN {X 0,Y 607.908,Z 965.052,A -85,B 0,C 180,E1 27612.861,E2 27612.861} C_VEL
LIN {X 0,Y 607.906,Z 951.242,A -85,B 0,C 180,E1 27610.898,E2 27610.898} C_VEL
LIN {X 0,Y 607.91,Z 936.609,A -85,B 0,C 180,E1 27609.093,E2 27609.093} C_VEL
LIN {X 0,Y 607.914,Z 920.209,A -85,B 0,C 180,E1 27607.323,E2 27607.323} C_VEL
LIN {X 0,Y 607.905,Z 902.853,A -85,B 0,C 180,E1 27605.67,E2 27605.67} C_VEL
LIN {X 0,Y 607.908,Z 884.653,A -85,B 0,C 180,E1 27604.164,E2 27604.164} C_VEL
LIN {X 0,Y 607.913,Z 864.226,A -85,B 0,C 180,E1 27602.689,E2 27602.689} C_VEL
LIN {X 0,Y 607.916,Z 844.862,A -85,B 0,C 180,E1 27601.476,E2 27601.476} C_VEL
LIN {X 0,Y 607.918,Z 824.382,A -85,B 0,C 180,E1 27600.384,E2 27600.384} C_VEL
LIN {X 0,Y 607.914,Z 805.451,A -85,B 0,C 180,E1 27599.523,E2 27599.523} C_VEL
LIN {X 0,Y 607.915,Z 783.158,A -85,B 0,C 180,E1 27598.69,E2 27598.69} C_VEL
LIN {X 0,Y 607.912,Z 764.555,A -85,B 0,C 180,E1 27598.136,E2 27598.136} C_VEL
LIN {X 0,Y 607.91,Z 742.804,A -85,B 0,C 180,E1 27597.636,E2 27597.636} C_VEL
LIN {X 0,Y 607.915,Z 700.32,A -85,B 0,C 180,E1 27597.014,E2 27597.014} C_VEL
LIN {X 0,Y 607.913,Z 490.035,A -85,B 0,C 180,E1 27594.063,E2 27594.063} C_VEL
LIN {X 0,Y 607.918,Z 390.77,A -85,B 0,C 180,E1 27592.618,E2 27592.618} C_VEL
LIN {X 0,Y 607.887,Z 355.818,A -85,B 0,C 180,E1 27590.252,E2 27590.252} C_VEL
LIN {X 0,Y 607.858,Z 355.316,A -85,B 0,C 180,E1 27589.978,E2 27589.978} C_VEL
LIN {X 0,Y 607.845,Z 355.324,A -85,B 0,C 180,E1 27587.191,E2 27587.191} C_VEL
LIN {X 0,Y 607.879,Z 355.326,A -85,B 0,C 180,E1 27584.051,E2 27584.051} C_VEL
LIN {X 0,Y 607.836,Z 355.326,A -85,B 0,C 180,E1 27581.145,E2 27581.145} C_VEL
LIN {X 0,Y 607.894,Z 355.328,A -85,B 0,C 180,E1 27578.021,E2 27578.021} C_VEL
LIN {X 0,Y 607.828,Z 355.325,A -85,B 0,C 180,E1 27575.151,E2 27575.151} C_VEL
LIN {X 0,Y 607.897,Z 355.327,A -85,B 0,C 180,E1 27572.202,E2 27572.202} C_VEL
LIN {X 0,Y 607.825,Z 355.327,A -85,B 0,C 180,E1 27569.137,E2 27569.137} C_VEL
LIN {X 0,Y 607.839,Z 355.328,A -85,B 0,C 180,E1 27566.473,E2 27566.473} C_VEL
LIN {X 0,Y 607.838,Z 355.327,A -85,B 0,C 180,E1 27563.15,E2 27563.15} C_VEL
LIN {X 0,Y 607.837,Z 355.327,A -85,B 0,C 180,E1 27560.409,E2 27560.409} C_VEL
LIN {X 0,Y 607.866,Z 355.326,A -85,B 0,C 180,E1 27557.222,E2 27557.222} C_VEL
LIN {X 0,Y 607.836,Z 355.326,A -85,B 0,C 180,E1 27554.351,E2 27554.351} C_VEL
LIN {X 0,Y 607.903,Z 355.324,A -85,B 0,C 180,E1 27551.287,E2 27551.287} C_VEL
LIN {X 0,Y 607.838,Z 355.326,A -85,B 0,C 180,E1 27548.323,E2 27548.323} C_VEL
LIN {X 0,Y 607.916,Z 355.325,A -85,B 0,C 180,E1 27545.284,E2 27545.284} C_VEL
LIN {X 0,Y 607.843,Z 355.325,A -85,B 0,C 180,E1 27542.262,E2 27542.262} C_VEL
LIN {X 0,Y 607.913,Z 355.328,A -85,B 0,C 180,E1 27539.246,E2 27539.246} C_VEL
LIN {X 0,Y 607.888,Z 355.322,A -85,B 0,C 180,E1 27536.676,E2 27536.676} C_VEL
LIN {X 0,Y 606.832,Z 355.454,A -85,B 0,C 180,E1 27535.95,E2 27535.95} C_VEL
LIN {X 0,Y 600.422,Z 356.251,A -85,B 0,C 180,E1 27533.914,E2 27533.914} C_VEL
LIN {X 0,Y 599.941,Z 356.315,A -85,B 0,C 180,E1 27533.384,E2 27533.384} C_VEL
LIN {X 0,Y 599.921,Z 356.312,A -85,B 0,C 180,E1 27530.115,E2 27530.115} C_VEL
LIN {X 0,Y 599.958,Z 356.316,A -85,B 0,C 180,E1 27527.096,E2 27527.096} C_VEL
LIN {X 0,Y 599.925,Z 356.311,A -85,B 0,C 180,E1 27523.939,E2 27523.939} C_VEL
LIN {X 0,Y 599.972,Z 356.317,A -85,B 0,C 180,E1 27520.834,E2 27520.834} C_VEL
LIN {X 0,Y 599.926,Z 356.311,A -85,B 0,C 180,E1 27517.654,E2 27517.654} C_VEL
LIN {X 0,Y 599.978,Z 356.314,A -85,B 0,C 180,E1 27514.535,E2 27514.535} C_VEL
LIN {X 0,Y 599.928,Z 356.311,A -85,B 0,C 180,E1 27511.424,E2 27511.424} C_VEL
LIN {X 0,Y 599.976,Z 356.314,A -85,B 0,C 180,E1 27508.335,E2 27508.335} C_VEL
LIN {X 0,Y 599.932,Z 356.311,A -85,B 0,C 180,E1 27505.242,E2 27505.242} C_VEL
LIN {X 0,Y 599.974,Z 356.314,A -85,B 0,C 180,E1 27502.171,E2 27502.171} C_VEL
LIN {X 0,Y 599.935,Z 356.31,A -85,B 0,C 180,E1 27499.017,E2 27499.017} C_VEL
LIN {X 0,Y 599.971,Z 356.311,A -85,B 0,C 180,E1 27495.845,E2 27495.845} C_VEL
LIN {X 0,Y 599.939,Z 356.311,A -85,B 0,C 180,E1 27492.695,E2 27492.695} C_VEL
LIN {X 0,Y 599.971,Z 356.309,A -85,B 0,C 180,E1 27489.534,E2 27489.534} C_VEL
LIN {X 0,Y 599.946,Z 356.312,A -85,B 0,C 180,E1 27486.387,E2 27486.387} C_VEL
LIN {X 0,Y 599.977,Z 356.306,A -85,B 0,C 180,E1 27483.13,E2 27483.13} C_VEL
LIN {X 0,Y 599.977,Z 356.314,A -85,B 0,C 180,E1 27479.772,E2 27479.772} C_VEL
LIN {X 0,Y 599.952,Z 356.308,A -85,B 0,C 180,E1 27476.498,E2 27476.498} C_VEL
LIN {X 0,Y 599.965,Z 356.312,A -85,B 0,C 180,E1 27473.327,E2 27473.327} C_VEL
LIN {X 0,Y 599.952,Z 356.309,A -85,B 0,C 180,E1 27470.177,E2 27470.177} C_VEL
LIN {X 0,Y 599.961,Z 356.311,A -85,B 0,C 180,E1 27467.053,E2 27467.053} C_VEL
LIN {X 0,Y 599.954,Z 356.311,A -85,B 0,C 180,E1 27463.883,E2 27463.883} C_VEL
LIN {X 0,Y 599.958,Z 356.311,A -85,B 0,C 180,E1 27460.755,E2 27460.755} C_VEL
LIN {X 0,Y 599.958,Z 356.29,A -85,B 0,C 180,E1 27457.563,E2 27457.563} C_VEL
LIN {X 0,Y 599.99,Z 356.42,A -85,B 0,C 180,E1 27456.264,E2 27456.264} C_VEL
LIN {X 0,Y 601.081,Z 360.007,A -85,B 0,C 180,E1 27455.917,E2 27455.917} C_VEL
LIN {X 0,Y 601.396,Z 362.791,A -85,B 0,C 180,E1 27455.77,E2 27455.77} C_VEL
LIN {X 0,Y 601.354,Z 509.563,A -85,B 0,C 180,E1 27453.63,E2 27453.63} C_VEL
LIN {X 0,Y 601.149,Z 709.774,A -85,B 0,C 180,E1 27450.781,E2 27450.781} C_VEL
LIN {X 0,Y 601.069,Z 733.34,A -85,B 0,C 180,E1 27450.26,E2 27450.26} C_VEL
LIN {X 0,Y 600.998,Z 753.673,A -85,B 0,C 180,E1 27449.652,E2 27449.652} C_VEL
LIN {X 0,Y 600.873,Z 775.98,A -85,B 0,C 180,E1 27448.806,E2 27448.806} C_VEL
LIN {X 0,Y 600.788,Z 796.567,A -85,B 0,C 180,E1 27447.852,E2 27447.852} C_VEL
LIN {X 0,Y 600.647,Z 818.129,A -85,B 0,C 180,E1 27446.658,E2 27446.658} C_VEL
LIN {X 0,Y 600.543,Z 838.165,A -85,B 0,C 180,E1 27445.366,E2 27445.366} C_VEL
LIN {X 0,Y 600.417,Z 857.883,A -85,B 0,C 180,E1 27443.88,E2 27443.88} C_VEL
LIN {X 0,Y 600.287,Z 876.854,A -85,B 0,C 180,E1 27442.244,E2 27442.244} C_VEL
LIN {X 0,Y 600.209,Z 894.467,A -85,B 0,C 180,E1 27440.505,E2 27440.505} C_VEL
LIN {X 0,Y 600.117,Z 909.858,A -85,B 0,C 180,E1 27438.757,E2 27438.757} C_VEL
LIN {X 0,Y 600.039,Z 925.011,A -85,B 0,C 180,E1 27436.802,E2 27436.802} C_VEL
LIN {X 0,Y 599.994,Z 937.612,A -85,B 0,C 180,E1 27434.93,E2 27434.93} C_VEL
LIN {X 0,Y 599.953,Z 949.711,A -85,B 0,C 180,E1 27432.842,E2 27432.842} C_VEL
LIN {X 0,Y 599.948,Z 959.345,A -85,B 0,C 180,E1 27430.9,E2 27430.9} C_VEL
LIN {X 0,Y 599.91,Z 968.039,A -85,B 0,C 180,E1 27428.795,E2 27428.795} C_VEL
LIN {X 0,Y 599.912,Z 974.678,A -85,B 0,C 180,E1 27426.836,E2 27426.836} C_VEL
LIN {X 0,Y 599.912,Z 980.545,A -85,B 0,C 180,E1 27424.601,E2 27424.601} C_VEL
LIN {X 0,Y 599.884,Z 984.329,A -85,B 0,C 180,E1 27422.61,E2 27422.61} C_VEL
LIN {X 0,Y 599.9,Z 987.001,A -85,B 0,C 180,E1 27420.328,E2 27420.328} C_VEL
LIN {X 0,Y 599.898,Z 987.921,A -85,B 0,C 180,E1 27418.329,E2 27418.329} C_VEL
LIN {X 0,Y 599.881,Z 987.367,A -85,B 0,C 180,E1 27416.104,E2 27416.104} C_VEL
LIN {X 0,Y 599.914,Z 985.58,A -85,B 0,C 180,E1 27414.195,E2 27414.195} C_VEL
LIN {X 0,Y 599.891,Z 981.77,A -85,B 0,C 180,E1 27411.878,E2 27411.878} C_VEL
LIN {X 0,Y 599.9,Z 977.191,A -85,B 0,C 180,E1 27409.956,E2 27409.956} C_VEL
LIN {X 0,Y 599.925,Z 970.297,A -85,B 0,C 180,E1 27407.731,E2 27407.731} C_VEL
LIN {X 0,Y 599.911,Z 962.708,A -85,B 0,C 180,E1 27405.781,E2 27405.781} C_VEL
LIN {X 0,Y 599.948,Z 952.896,A -85,B 0,C 180,E1 27403.672,E2 27403.672} C_VEL
LIN {X 0,Y 599.989,Z 942.603,A -85,B 0,C 180,E1 27401.804,E2 27401.804} C_VEL
LIN {X 0,Y 600.04,Z 929.317,A -85,B 0,C 180,E1 27399.72,E2 27399.72} C_VEL
LIN {X 0,Y 600.091,Z 915.292,A -85,B 0,C 180,E1 27397.818,E2 27397.818} C_VEL
LIN {X 0,Y 600.179,Z 899.307,A -85,B 0,C 180,E1 27395.937,E2 27395.937} C_VEL
LIN {X 0,Y 600.276,Z 881.961,A -85,B 0,C 180,E1 27394.148,E2 27394.148} C_VEL
LIN {X 0,Y 600.375,Z 863.524,A -85,B 0,C 180,E1 27392.486,E2 27392.486} C_VEL
LIN {X 0,Y 600.492,Z 843.913,A -85,B 0,C 180,E1 27390.961,E2 27390.961} C_VEL
LIN {X 0,Y 600.628,Z 823.458,A -85,B 0,C 180,E1 27389.576,E2 27389.576} C_VEL
LIN {X 0,Y 600.728,Z 803.614,A -85,B 0,C 180,E1 27388.426,E2 27388.426} C_VEL
LIN {X 0,Y 600.866,Z 781.402,A -85,B 0,C 180,E1 27387.34,E2 27387.34} C_VEL
LIN {X 0,Y 600.947,Z 761.523,A -85,B 0,C 180,E1 27386.534,E2 27386.534} C_VEL
LIN {X 0,Y 601.057,Z 738.111,A -85,B 0,C 180,E1 27385.779,E2 27385.779} C_VEL
LIN {X 0,Y 601.118,Z 717.605,A -85,B 0,C 180,E1 27385.281,E2 27385.281} C_VEL
LIN {X 0,Y 601.178,Z 689.502,A -85,B 0,C 180,E1 27384.82,E2 27384.82} C_VEL
LIN {X 0,Y 601.414,Z 477.951,A -85,B 0,C 180,E1 27381.827,E2 27381.827} C_VEL
LIN {X 0,Y 601.382,Z 362.673,A -85,B 0,C 180,E1 27380.137,E2 27380.137} C_VEL
LIN {X 0,Y 601.098,Z 359.616,A -85,B 0,C 180,E1 27379.966,E2 27379.966} C_VEL
LIN {X 0,Y 599.996,Z 356.472,A -85,B 0,C 180,E1 27379.603,E2 27379.603} C_VEL
LIN {X 0,Y 599.975,Z 356.311,A -85,B 0,C 180,E1 27376.358,E2 27376.358} C_VEL
LIN {X 0,Y 599.955,Z 356.308,A -85,B 0,C 180,E1 27373.1,E2 27373.1} C_VEL
LIN {X 0,Y 599.964,Z 356.314,A -85,B 0,C 180,E1 27369.96,E2 27369.96} C_VEL
LIN {X 0,Y 599.957,Z 356.31,A -85,B 0,C 180,E1 27366.796,E2 27366.796} C_VEL
LIN {X 0,Y 599.955,Z 356.311,A -85,B 0,C 180,E1 27363.631,E2 27363.631} C_VEL
LIN {X 0,Y 599.963,Z 356.312,A -85,B 0,C 180,E1 27360.478,E2 27360.478} C_VEL
LIN {X 0,Y 599.95,Z 356.309,A -85,B 0,C 180,E1 27357.326,E2 27357.326} C_VEL
LIN {X 0,Y 599.972,Z 356.317,A -85,B 0,C 180,E1 27354.07,E2 27354.07} C_VEL
LIN {X 0,Y 599.968,Z 356.307,A -85,B 0,C 180,E1 27350.794,E2 27350.794} C_VEL
LIN {X 0,Y 599.943,Z 356.314,A -85,B 0,C 180,E1 27347.585,E2 27347.585} C_VEL
LIN {X 0,Y 599.975,Z 356.309,A -85,B 0,C 180,E1 27344.418,E2 27344.418} C_VEL
LIN {X 0,Y 599.925,Z 356.313,A -85,B 0,C 180,E1 27341.237,E2 27341.237} C_VEL
LIN {X 0,Y 599.977,Z 356.313,A -85,B 0,C 180,E1 27338.081,E2 27338.081} C_VEL
LIN {X 0,Y 599.915,Z 356.314,A -85,B 0,C 180,E1 27335.05,E2 27335.05} C_VEL
LIN {X 0,Y 599.979,Z 356.313,A -85,B 0,C 180,E1 27331.969,E2 27331.969} C_VEL
LIN {X 0,Y 599.903,Z 356.315,A -85,B 0,C 180,E1 27328.891,E2 27328.891} C_VEL
LIN {X 0,Y 599.979,Z 356.315,A -85,B 0,C 180,E1 27325.833,E2 27325.833} C_VEL
LIN {X 0,Y 599.892,Z 356.316,A -85,B 0,C 180,E1 27322.77,E2 27322.77} C_VEL
LIN {X 0,Y 599.968,Z 356.317,A -85,B 0,C 180,E1 27319.714,E2 27319.714} C_VEL
LIN {X 0,Y 599.89,Z 356.317,A -85,B 0,C 180,E1 27316.612,E2 27316.612} C_VEL
LIN {X 0,Y 599.971,Z 356.316,A -85,B 0,C 180,E1 27313.627,E2 27313.627} C_VEL
LIN {X 0,Y 599.902,Z 356.302,A -85,B 0,C 180,E1 27310.535,E2 27310.535} C_VEL
LIN {X 0,Y 599.99,Z 356.848,A -85,B 0,C 180,E1 27310.307,E2 27310.307} C_VEL
LIN {X 0,Y 601.27,Z 360.468,A -85,B 0,C 180,E1 27309.934,E2 27309.934} C_VEL
LIN {X 0,Y 601.281,Z 391.488,A -85,B 0,C 180,E1 27307.845,E2 27307.845} C_VEL
LIN {X 0,Y 601.544,Z 396.244,A -85,B 0,C 180,E1 27307.753,E2 27307.753} C_VEL
LIN {X 0,Y 601.307,Z 602.693,A -85,B 0,C 180,E1 27304.774,E2 27304.774} C_VEL
LIN {X 0,Y 601.148,Z 739.245,A -85,B 0,C 180,E1 27302.833,E2 27302.833} C_VEL
LIN {X 0,Y 601.067,Z 762.966,A -85,B 0,C 180,E1 27302.313,E2 27302.313} C_VEL
LIN {X 0,Y 601.001,Z 782.313,A -85,B 0,C 180,E1 27301.74,E2 27301.74} C_VEL
LIN {X 0,Y 600.876,Z 805.215,A -85,B 0,C 180,E1 27300.883,E2 27300.883} C_VEL
LIN {X 0,Y 600.793,Z 824.268,A -85,B 0,C 180,E1 27300.008,E2 27300.008} C_VEL
LIN {X 0,Y 600.656,Z 845.442,A -85,B 0,C 180,E1 27298.866,E2 27298.866} C_VEL
LIN {X 0,Y 600.556,Z 864.867,A -85,B 0,C 180,E1 27297.631,E2 27297.631} C_VEL
LIN {X 0,Y 600.417,Z 884.954,A -85,B 0,C 180,E1 27296.159,E2 27296.159} C_VEL
LIN {X 0,Y 600.324,Z 903.725,A -85,B 0,C 180,E1 27294.581,E2 27294.581} C_VEL
LIN {X 0,Y 600.228,Z 921.026,A -85,B 0,C 180,E1 27292.901,E2 27292.901} C_VEL
LIN {X 0,Y 600.13,Z 938.269,A -85,B 0,C 180,E1 27290.992,E2 27290.992} C_VEL
LIN {X 0,Y 600.066,Z 952.978,A -85,B 0,C 180,E1 27289.134,E2 27289.134} C_VEL
LIN {X 0,Y 600.009,Z 966.435,A -85,B 0,C 180,E1 27287.157,E2 27287.157} C_VEL
LIN {X 0,Y 599.973,Z 978.738,A -85,B 0,C 180,E1 27285.071,E2 27285.071} C_VEL
LIN {X 0,Y 599.926,Z 988.137,A -85,B 0,C 180,E1 27283.201,E2 27283.201} C_VEL
LIN {X 0,Y 599.905,Z 997.26,A -85,B 0,C 180,E1 27281.052,E2 27281.052} C_VEL
LIN {X 0,Y 599.919,Z 1003.946,A -85,B 0,C 180,E1 27279.112,E2 27279.112} C_VEL
LIN {X 0,Y 599.885,Z 1009.802,A -85,B 0,C 180,E1 27276.991,E2 27276.991} C_VEL
LIN {X 0,Y 599.906,Z 1013.794,A -85,B 0,C 180,E1 27274.974,E2 27274.974} C_VEL
LIN {X 0,Y 599.892,Z 1016.627,A -85,B 0,C 180,E1 27272.868,E2 27272.868} C_VEL
LIN {X 0,Y 599.884,Z 1017.827,A -85,B 0,C 180,E1 27270.766,E2 27270.766} C_VEL
LIN {X 0,Y 599.915,Z 1017.694,A -85,B 0,C 180,E1 27268.666,E2 27268.666} C_VEL
LIN {X 0,Y 599.886,Z 1015.957,A -85,B 0,C 180,E1 27266.563,E2 27266.563} C_VEL
LIN {X 0,Y 599.9,Z 1013.006,A -85,B 0,C 180,E1 27264.551,E2 27264.551} C_VEL
LIN {X 0,Y 599.914,Z 1008.087,A -85,B 0,C 180,E1 27262.341,E2 27262.341} C_VEL
LIN {X 0,Y 599.893,Z 1002.437,A -85,B 0,C 180,E1 27260.408,E2 27260.408} C_VEL
LIN {X 0,Y 599.929,Z 994.161,A -85,B 0,C 180,E1 27258.174,E2 27258.174} C_VEL
LIN {X 0,Y 599.935,Z 985.842,A -85,B 0,C 180,E1 27256.314,E2 27256.314} C_VEL
LIN {X 0,Y 599.967,Z 974.313,A -85,B 0,C 180,E1 27254.142,E2 27254.142} C_VEL
LIN {X 0,Y 600.009,Z 962.61,A -85,B 0,C 180,E1 27252.248,E2 27252.248} C_VEL
LIN {X 0,Y 600.079,Z 948.551,A -85,B 0,C 180,E1 27250.288,E2 27250.288} C_VEL
LIN {X 0,Y 600.163,Z 933.087,A -85,B 0,C 180,E1 27248.4,E2 27248.4} C_VEL
LIN {X 0,Y 600.238,Z 917.111,A -85,B 0,C 180,E1 27246.699,E2 27246.699} C_VEL
LIN {X 0,Y 600.348,Z 899.252,A -85,B 0,C 180,E1 27245.03,E2 27245.03} C_VEL
LIN {X 0,Y 600.47,Z 880.65,A -85,B 0,C 180,E1 27243.5,E2 27243.5} C_VEL
LIN {X 0,Y 600.566,Z 861.019,A -85,B 0,C 180,E1 27242.111,E2 27242.111} C_VEL
LIN {X 0,Y 600.709,Z 839.866,A -85,B 0,C 180,E1 27240.815,E2 27240.815} C_VEL
LIN {X 0,Y 600.801,Z 819.801,A -85,B 0,C 180,E1 27239.772,E2 27239.772} C_VEL
LIN {X 0,Y 600.932,Z 797.647,A -85,B 0,C 180,E1 27238.812,E2 27238.812} C_VEL
LIN {X 0,Y 601.009,Z 777.778,A -85,B 0,C 180,E1 27238.113,E2 27238.113} C_VEL
LIN {X 0,Y 601.106,Z 754.497,A -85,B 0,C 180,E1 27237.477,E2 27237.477} C_VEL
LIN {X 0,Y 601.153,Z 734.897,A -85,B 0,C 180,E1 27237.095,E2 27237.095} C_VEL
LIN {X 0,Y 601.403,Z 510.296,A -85,B 0,C 180,E1 27233.905,E2 27233.905} C_VEL
LIN {X 0,Y 601.373,Z 391.971,A -85,B 0,C 180,E1 27232.171,E2 27232.171} C_VEL
LIN {X 0,Y 601.163,Z 388.311,A -85,B 0,C 180,E1 27231.964,E2 27231.964} C_VEL
LIN {X 0,Y 601.106,Z 359.613,A -85,B 0,C 180,E1 27229.994,E2 27229.994} C_VEL
LIN {X 0,Y 599.929,Z 356.497,A -85,B 0,C 180,E1 27229.632,E2 27229.632} C_VEL
LIN {X 0,Y 599.919,Z 356.311,A -85,B 0,C 180,E1 27227.025,E2 27227.025} C_VEL
LIN {X 0,Y 599.911,Z 356.312,A -85,B 0,C 180,E1 27223.762,E2 27223.762} C_VEL
LIN {X 0,Y 599.905,Z 356.316,A -85,B 0,C 180,E1 27220.98,E2 27220.98} C_VEL
LIN {X 0,Y 599.913,Z 356.317,A -85,B 0,C 180,E1 27217.665,E2 27217.665} C_VEL
LIN {X 0,Y 599.894,Z 356.312,A -85,B 0,C 180,E1 27214.92,E2 27214.92} C_VEL
LIN {X 0,Y 599.94,Z 356.315,A -85,B 0,C 180,E1 27211.779,E2 27211.779} C_VEL
LIN {X 0,Y 599.884,Z 356.316,A -85,B 0,C 180,E1 27208.959,E2 27208.959} C_VEL
LIN {X 0,Y 599.955,Z 356.317,A -85,B 0,C 180,E1 27205.995,E2 27205.995} C_VEL
LIN {X 0,Y 599.889,Z 356.316,A -85,B 0,C 180,E1 27202.955,E2 27202.955} C_VEL
LIN {X 0,Y 599.916,Z 356.316,A -85,B 0,C 180,E1 27200.181,E2 27200.181} C_VEL
LIN {X 0,Y 599.902,Z 356.315,A -85,B 0,C 180,E1 27196.94,E2 27196.94} C_VEL
LIN {X 0,Y 599.907,Z 356.315,A -85,B 0,C 180,E1 27194.182,E2 27194.182} C_VEL
LIN {X 0,Y 599.913,Z 356.314,A -85,B 0,C 180,E1 27190.855,E2 27190.855} C_VEL
LIN {X 0,Y 599.909,Z 356.315,A -85,B 0,C 180,E1 27188.048,E2 27188.048} C_VEL
LIN {X 0,Y 599.925,Z 356.313,A -85,B 0,C 180,E1 27184.747,E2 27184.747} C_VEL
LIN {X 0,Y 599.912,Z 356.315,A -85,B 0,C 180,E1 27181.91,E2 27181.91} C_VEL
LIN {X 0,Y 599.94,Z 356.312,A -85,B 0,C 180,E1 27178.663,E2 27178.663} C_VEL
LIN {X 0,Y 599.918,Z 356.315,A -85,B 0,C 180,E1 27175.698,E2 27175.698} C_VEL
LIN {X 0,Y 599.941,Z 356.315,A -85,B 0,C 180,E1 27173.384,E2 27173.384} C_VEL
LIN {X 0,Y 599.005,Z 356.438,A -85,B 0,C 180,E1 27172.648,E2 27172.648} C_VEL
LIN {X 0,Y 592.436,Z 357.248,A -85,B 0,C 180,E1 27170.531,E2 27170.531} C_VEL
LIN {X 0,Y 591.979,Z 357.301,A -85,B 0,C 180,E1 27170.047,E2 27170.047} C_VEL
LIN {X 0,Y 592.027,Z 357.305,A -85,B 0,C 180,E1 27167.007,E2 27167.007} C_VEL
LIN {X 0,Y 591.982,Z 357.3,A -85,B 0,C 180,E1 27163.818,E2 27163.818} C_VEL
LIN {X 0,Y 592.038,Z 357.303,A -85,B 0,C 180,E1 27160.732,E2 27160.732} C_VEL
LIN {X 0,Y 591.985,Z 357.301,A -85,B 0,C 180,E1 27157.56,E2 27157.56} C_VEL
LIN {X 0,Y 592.039,Z 357.302,A -85,B 0,C 180,E1 27154.491,E2 27154.491} C_VEL
LIN {X 0,Y 591.988,Z 357.301,A -85,B 0,C 180,E1 27151.336,E2 27151.336} C_VEL
LIN {X 0,Y 592.036,Z 357.301,A -85,B 0,C 180,E1 27148.202,E2 27148.202} C_VEL
LIN {X 0,Y 591.992,Z 357.301,A -85,B 0,C 180,E1 27145.071,E2 27145.071} C_VEL
LIN {X 0,Y 592.036,Z 357.298,A -85,B 0,C 180,E1 27141.9,E2 27141.9} C_VEL
LIN {X 0,Y 592.001,Z 357.301,A -85,B 0,C 180,E1 27138.721,E2 27138.721} C_VEL
LIN {X 0,Y 592.033,Z 357.296,A -85,B 0,C 180,E1 27135.449,E2 27135.449} C_VEL
LIN {X 0,Y 592.028,Z 357.305,A -85,B 0,C 180,E1 27132.148,E2 27132.148} C_VEL
LIN {X 0,Y 592.007,Z 357.298,A -85,B 0,C 180,E1 27128.867,E2 27128.867} C_VEL
LIN {X 0,Y 592.03,Z 357.301,A -85,B 0,C 180,E1 27125.633,E2 27125.633} C_VEL
LIN {X 0,Y 592.006,Z 357.3,A -85,B 0,C 180,E1 27122.481,E2 27122.481} C_VEL
LIN {X 0,Y 592.027,Z 357.299,A -85,B 0,C 180,E1 27119.322,E2 27119.322} C_VEL
LIN {X 0,Y 592.012,Z 357.3,A -85,B 0,C 180,E1 27116.152,E2 27116.152} C_VEL
LIN {X 0,Y 592.033,Z 357.295,A -85,B 0,C 180,E1 27112.854,E2 27112.854} C_VEL
LIN {X 0,Y 592.036,Z 357.305,A -85,B 0,C 180,E1 27109.532,E2 27109.532} C_VEL
LIN {X 0,Y 592.022,Z 357.297,A -85,B 0,C 180,E1 27106.278,E2 27106.278} C_VEL
LIN {X 0,Y 592.022,Z 357.292,A -85,B 0,C 180,E1 27103.077,E2 27103.077} C_VEL
LIN {X 0,Y 592.019,Z 357.301,A -85,B 0,C 180,E1 27099.917,E2 27099.917} C_VEL
LIN {X 0,Y 592.017,Z 357.275,A -85,B 0,C 180,E1 27096.811,E2 27096.811} C_VEL
LIN {X 0,Y 593.151,Z 360.471,A -85,B 0,C 180,E1 27096.482,E2 27096.482} C_VEL
LIN {X 0,Y 594.489,Z 363.175,A -85,B 0,C 180,E1 27096.283,E2 27096.283} C_VEL
LIN {X 0,Y 595.21,Z 365.986,A -85,B 0,C 180,E1 27096.186,E2 27096.186} C_VEL
LIN {X 0,Y 594.733,Z 572.073,A -85,B 0,C 180,E1 27093.179,E2 27093.179} C_VEL
LIN {X 0,Y 594.416,Z 710.235,A -85,B 0,C 180,E1 27091.193,E2 27091.193} C_VEL
LIN {X 0,Y 594.252,Z 733.717,A -85,B 0,C 180,E1 27090.666,E2 27090.666} C_VEL
LIN {X 0,Y 594.106,Z 754.954,A -85,B 0,C 180,E1 27090.022,E2 27090.022} C_VEL
LIN {X 0,Y 593.859,Z 776.741,A -85,B 0,C 180,E1 27089.178,E2 27089.178} C_VEL
LIN {X 0,Y 593.672,Z 798.233,A -85,B 0,C 180,E1 27088.164,E2 27088.164} C_VEL
LIN {X 0,Y 593.392,Z 819.532,A -85,B 0,C 180,E1 27086.955,E2 27086.955} C_VEL
LIN {X 0,Y 593.157,Z 840.061,A -85,B 0,C 180,E1 27085.599,E2 27085.599} C_VEL
LIN {X 0,Y 592.926,Z 859.592,A -85,B 0,C 180,E1 27084.093,E2 27084.093} C_VEL
LIN {X 0,Y 592.673,Z 878.318,A -85,B 0,C 180,E1 27082.436,E2 27082.436} C_VEL
LIN {X 0,Y 592.499,Z 895.74,A -85,B 0,C 180,E1 27080.675,E2 27080.675} C_VEL
LIN {X 0,Y 592.334,Z 911.013,A -85,B 0,C 180,E1 27078.903,E2 27078.903} C_VEL
LIN {X 0,Y 592.182,Z 925.984,A -85,B 0,C 180,E1 27076.921,E2 27076.921} C_VEL
LIN {X 0,Y 592.091,Z 939.124,A -85,B 0,C 180,E1 27074.924,E2 27074.924} C_VEL
LIN {X 0,Y 592.012,Z 950.429,A -85,B 0,C 180,E1 27072.908,E2 27072.908} C_VEL
LIN {X 0,Y 591.982,Z 960.308,A -85,B 0,C 180,E1 27070.871,E2 27070.871} C_VEL
LIN {X 0,Y 591.926,Z 968.536,A -85,B 0,C 180,E1 27068.807,E2 27068.807} C_VEL
LIN {X 0,Y 591.909,Z 975.432,A -85,B 0,C 180,E1 27066.715,E2 27066.715} C_VEL
LIN {X 0,Y 591.915,Z 980.761,A -85,B 0,C 180,E1 27064.591,E2 27064.591} C_VEL
LIN {X 0,Y 591.883,Z 984.736,A -85,B 0,C 180,E1 27062.426,E2 27062.426} C_VEL
LIN {X 0,Y 591.893,Z 987.1,A -85,B 0,C 180,E1 27060.22,E2 27060.22} C_VEL
LIN {X 0,Y 591.904,Z 987.958,A -85,B 0,C 180,E1 27058.177,E2 27058.177} C_VEL
LIN {X 0,Y 591.881,Z 987.316,A -85,B 0,C 180,E1 27056.001,E2 27056.001} C_VEL
LIN {X 0,Y 591.907,Z 985.408,A -85,B 0,C 180,E1 27053.994,E2 27053.994} C_VEL
LIN {X 0,Y 591.905,Z 981.54,A -85,B 0,C 180,E1 27051.686,E2 27051.686} C_VEL
LIN {X 0,Y 591.895,Z 977.01,A -85,B 0,C 180,E1 27049.778,E2 27049.778} C_VEL
LIN {X 0,Y 591.935,Z 969.947,A -85,B 0,C 180,E1 27047.493,E2 27047.493} C_VEL
LIN {X 0,Y 591.946,Z 962.21,A -85,B 0,C 180,E1 27045.493,E2 27045.493} C_VEL
LIN {X 0,Y 591.998,Z 951.903,A -85,B 0,C 180,E1 27043.285,E2 27043.285} C_VEL
LIN {X 0,Y 592.071,Z 941.701,A -85,B 0,C 180,E1 27041.425,E2 27041.425} C_VEL
LIN {X 0,Y 592.188,Z 928.476,A -85,B 0,C 180,E1 27039.348,E2 27039.348} C_VEL
LIN {X 0,Y 592.318,Z 914.39,A -85,B 0,C 180,E1 27037.423,E2 27037.423} C_VEL
LIN {X 0,Y 592.457,Z 898.681,A -85,B 0,C 180,E1 27035.565,E2 27035.565} C_VEL
LIN {X 0,Y 592.668,Z 880.823,A -85,B 0,C 180,E1 27033.714,E2 27033.714} C_VEL
LIN {X 0,Y 592.904,Z 862.216,A -85,B 0,C 180,E1 27032.03,E2 27032.03} C_VEL
LIN {X 0,Y 593.102,Z 842.538,A -85,B 0,C 180,E1 27030.493,E2 27030.493} C_VEL
LIN {X 0,Y 593.377,Z 821.678,A -85,B 0,C 180,E1 27029.087,E2 27029.087} C_VEL
LIN {X 0,Y 593.609,Z 801.575,A -85,B 0,C 180,E1 27027.921,E2 27027.921} C_VEL
LIN {X 0,Y 593.846,Z 779.895,A -85,B 0,C 180,E1 27026.872,E2 27026.872} C_VEL
LIN {X 0,Y 594.062,Z 758.267,A -85,B 0,C 180,E1 27026.002,E2 27026.002} C_VEL
LIN {X 0,Y 594.242,Z 735.827,A -85,B 0,C 180,E1 27025.301,E2 27025.301} C_VEL
LIN {X 0,Y 594.388,Z 713.4,A -85,B 0,C 180,E1 27024.773,E2 27024.773} C_VEL
LIN {X 0,Y 594.507,Z 673.265,A -85,B 0,C 180,E1 27024.169,E2 27024.169} C_VEL
LIN {X 0,Y 594.982,Z 462.811,A -85,B 0,C 180,E1 27021.151,E2 27021.151} C_VEL
LIN {X 0,Y 595.04,Z 364.472,A -85,B 0,C 180,E1 27019.689,E2 27019.689} C_VEL
LIN {X 0,Y 593.473,Z 360.993,A -85,B 0,C 180,E1 27019.487,E2 27019.487} C_VEL
LIN {X 0,Y 592.03,Z 357.49,A -85,B 0,C 180,E1 27019.075,E2 27019.075} C_VEL
LIN {X 0,Y 592.027,Z 357.289,A -85,B 0,C 180,E1 27015.979,E2 27015.979} C_VEL
LIN {X 0,Y 592.012,Z 357.3,A -85,B 0,C 180,E1 27012.783,E2 27012.783} C_VEL
LIN {X 0,Y 592.025,Z 357.299,A -85,B 0,C 180,E1 27009.625,E2 27009.625} C_VEL
LIN {X 0,Y 592.027,Z 357.304,A -85,B 0,C 180,E1 27006.4,E2 27006.4} C_VEL
LIN {X 0,Y 592.033,Z 357.296,A -85,B 0,C 180,E1 27003.098,E2 27003.098} C_VEL
LIN {X 0,Y 592.018,Z 357.303,A -85,B 0,C 180,E1 26999.807,E2 26999.807} C_VEL
LIN {X 0,Y 592.029,Z 357.298,A -85,B 0,C 180,E1 26996.612,E2 26996.612} C_VEL
LIN {X 0,Y 592.004,Z 357.3,A -85,B 0,C 180,E1 26993.405,E2 26993.405} C_VEL
LIN {X 0,Y 592.031,Z 357.302,A -85,B 0,C 180,E1 26990.277,E2 26990.277} C_VEL
LIN {X 0,Y 591.997,Z 357.3,A -85,B 0,C 180,E1 26987.118,E2 26987.118} C_VEL
LIN {X 0,Y 592.034,Z 357.306,A -85,B 0,C 180,E1 26983.921,E2 26983.921} C_VEL
LIN {X 0,Y 591.999,Z 357.3,A -85,B 0,C 180,E1 26980.758,E2 26980.758} C_VEL
LIN {X 0,Y 591.995,Z 357.304,A -85,B 0,C 180,E1 26977.456,E2 26977.456} C_VEL
LIN {X 0,Y 592.009,Z 357.301,A -85,B 0,C 180,E1 26974.383,E2 26974.383} C_VEL
LIN {X 0,Y 591.978,Z 357.304,A -85,B 0,C 180,E1 26971.226,E2 26971.226} C_VEL
LIN {X 0,Y 591.991,Z 357.303,A -85,B 0,C 180,E1 26968.314,E2 26968.314} C_VEL
LIN {X 0,Y 591.966,Z 357.306,A -85,B 0,C 180,E1 26965.07,E2 26965.07} C_VEL
LIN {X 0,Y 591.978,Z 357.305,A -85,B 0,C 180,E1 26962.186,E2 26962.186} C_VEL
LIN {X 0,Y 591.956,Z 357.307,A -85,B 0,C 180,E1 26958.925,E2 26958.925} C_VEL
LIN {X 0,Y 591.982,Z 357.308,A -85,B 0,C 180,E1 26956.016,E2 26956.016} C_VEL
LIN {X 0,Y 591.964,Z 357.299,A -85,B 0,C 180,E1 26952.767,E2 26952.767} C_VEL
LIN {X 0,Y 592.016,Z 357.507,A -85,B 0,C 180,E1 26950.944,E2 26950.944} C_VEL
LIN {X 0,Y 593.381,Z 360.936,A -85,B 0,C 180,E1 26950.541,E2 26950.541} C_VEL
LIN {X 0,Y 594.658,Z 364.048,A -85,B 0,C 180,E1 26950.217,E2 26950.217} C_VEL
LIN {X 0,Y 594.555,Z 391.484,A -85,B 0,C 180,E1 26948.351,E2 26948.351} C_VEL
LIN {X 0,Y 595.214,Z 395.838,A -85,B 0,C 180,E1 26948.233,E2 26948.233} C_VEL
LIN {X 0,Y 594.732,Z 602.463,A -85,B 0,C 180,E1 26945.219,E2 26945.219} C_VEL
LIN {X 0,Y 594.413,Z 739.46,A -85,B 0,C 180,E1 26943.249,E2 26943.249} C_VEL
LIN {X 0,Y 594.251,Z 763.128,A -85,B 0,C 180,E1 26942.726,E2 26942.726} C_VEL
LIN {X 0,Y 594.113,Z 782.983,A -85,B 0,C 180,E1 26942.13,E2 26942.13} C_VEL
LIN {X 0,Y 593.861,Z 806.363,A -85,B 0,C 180,E1 26941.238,E2 26941.238} C_VEL
LIN {X 0,Y 593.682,Z 826.508,A -85,B 0,C 180,E1 26940.294,E2 26940.294} C_VEL
LIN {X 0,Y 593.399,Z 848.115,A -85,B 0,C 180,E1 26939.087,E2 26939.087} C_VEL
LIN {X 0,Y 593.194,Z 868.454,A -85,B 0,C 180,E1 26937.76,E2 26937.76} C_VEL
LIN {X 0,Y 592.93,Z 887.235,A -85,B 0,C 180,E1 26936.329,E2 26936.329} C_VEL
LIN {X 0,Y 592.699,Z 906.325,A -85,B 0,C 180,E1 26934.67,E2 26934.67} C_VEL
LIN {X 0,Y 592.538,Z 923.319,A -85,B 0,C 180,E1 26932.978,E2 26932.978} C_VEL
LIN {X 0,Y 592.352,Z 939.122,A -85,B 0,C 180,E1 26931.177,E2 26931.177} C_VEL
LIN {X 0,Y 592.227,Z 953.603,A -85,B 0,C 180,E1 26929.308,E2 26929.308} C_VEL
LIN {X 0,Y 592.12,Z 966.436,A -85,B 0,C 180,E1 26927.393,E2 26927.393} C_VEL
LIN {X 0,Y 592.03,Z 978.74,A -85,B 0,C 180,E1 26925.278,E2 26925.278} C_VEL
LIN {X 0,Y 591.962,Z 988.185,A -85,B 0,C 180,E1 26923.372,E2 26923.372} C_VEL
LIN {X 0,Y 591.927,Z 997.26,A -85,B 0,C 180,E1 26921.203,E2 26921.203} C_VEL
LIN {X 0,Y 591.918,Z 1003.946,A -85,B 0,C 180,E1 26919.237,E2 26919.237} C_VEL
LIN {X 0,Y 591.888,Z 1009.802,A -85,B 0,C 180,E1 26917.086,E2 26917.086} C_VEL
LIN {X 0,Y 591.909,Z 1013.794,A -85,B 0,C 180,E1 26915.042,E2 26915.042} C_VEL
LIN {X 0,Y 591.89,Z 1016.628,A -85,B 0,C 180,E1 26912.907,E2 26912.907} C_VEL
LIN {X 0,Y 591.884,Z 1017.827,A -85,B 0,C 180,E1 26910.777,E2 26910.777} C_VEL
LIN {X 0,Y 591.914,Z 1017.694,A -85,B 0,C 180,E1 26908.647,E2 26908.647} C_VEL
LIN {X 0,Y 591.888,Z 1015.957,A -85,B 0,C 180,E1 26906.516,E2 26906.516} C_VEL
LIN {X 0,Y 591.899,Z 1013.006,A -85,B 0,C 180,E1 26904.477,E2 26904.477} C_VEL
LIN {X 0,Y 591.925,Z 1008.088,A -85,B 0,C 180,E1 26902.237,E2 26902.237} C_VEL
LIN {X 0,Y 591.903,Z 1002.438,A -85,B 0,C 180,E1 26900.278,E2 26900.278} C_VEL
LIN {X 0,Y 591.952,Z 994.162,A -85,B 0,C 180,E1 26898.012,E2 26898.012} C_VEL
LIN {X 0,Y 591.987,Z 985.844,A -85,B 0,C 180,E1 26896.126,E2 26896.126} C_VEL
LIN {X 0,Y 592.053,Z 974.315,A -85,B 0,C 180,E1 26893.924,E2 26893.924} C_VEL
LIN {X 0,Y 592.133,Z 962.612,A -85,B 0,C 180,E1 26892.004,E2 26892.004} C_VEL
LIN {X 0,Y 592.253,Z 948.911,A -85,B 0,C 180,E1 26890.064,E2 26890.064} C_VEL
LIN {X 0,Y 592.42,Z 933.633,A -85,B 0,C 180,E1 26888.165,E2 26888.165} C_VEL
LIN {X 0,Y 592.568,Z 917.617,A -85,B 0,C 180,E1 26886.432,E2 26886.432} C_VEL
LIN {X 0,Y 592.795,Z 899.328,A -85,B 0,C 180,E1 26884.697,E2 26884.697} C_VEL
LIN {X 0,Y 593.043,Z 880.651,A -85,B 0,C 180,E1 26883.142,E2 26883.142} C_VEL
LIN {X 0,Y 593.241,Z 861.021,A -85,B 0,C 180,E1 26881.736,E2 26881.736} C_VEL
LIN {X 0,Y 593.526,Z 839.869,A -85,B 0,C 180,E1 26880.427,E2 26880.427} C_VEL
LIN {X 0,Y 593.716,Z 819.926,A -85,B 0,C 180,E1 26879.379,E2 26879.379} C_VEL
LIN {X 0,Y 593.98,Z 797.581,A -85,B 0,C 180,E1 26878.403,E2 26878.403} C_VEL
LIN {X 0,Y 594.134,Z 777.243,A -85,B 0,C 180,E1 26877.682,E2 26877.682} C_VEL
LIN {X 0,Y 594.331,Z 753.429,A -85,B 0,C 180,E1 26877.036,E2 26877.036} C_VEL
LIN {X 0,Y 594.427,Z 733.827,A -85,B 0,C 180,E1 26876.657,E2 26876.657} C_VEL
LIN {X 0,Y 594.926,Z 512.643,A -85,B 0,C 180,E1 26873.484,E2 26873.484} C_VEL
LIN {X 0,Y 595.051,Z 393.777,A -85,B 0,C 180,E1 26871.724,E2 26871.724} C_VEL
LIN {X 0,Y 594.438,Z 390.108,A -85,B 0,C 180,E1 26871.579,E2 26871.579} C_VEL
LIN {X 0,Y 594.61,Z 363.854,A -85,B 0,C 180,E1 26869.766,E2 26869.766} C_VEL
LIN {X 0,Y 592.039,Z 357.67,A -85,B 0,C 180,E1 26869.091,E2 26869.091} C_VEL
LIN {X 0,Y 592.03,Z 357.265,A -85,B 0,C 180,E1 26868.421,E2 26868.421} C_VEL
LIN {X 0,Y 591.96,Z 357.306,A -85,B 0,C 180,E1 26865.366,E2 26865.366} C_VEL
LIN {X 0,Y 592.031,Z 357.302,A -85,B 0,C 180,E1 26862.234,E2 26862.234} C_VEL
LIN {X 0,Y 591.955,Z 357.301,A -85,B 0,C 180,E1 26859.176,E2 26859.176} C_VEL
LIN {X 0,Y 592.036,Z 357.3,A -85,B 0,C 180,E1 26856.115,E2 26856.115} C_VEL
LIN {X 0,Y 591.95,Z 357.306,A -85,B 0,C 180,E1 26853.064,E2 26853.064} C_VEL
LIN {X 0,Y 592.033,Z 357.3,A -85,B 0,C 180,E1 26849.968,E2 26849.968} C_VEL
LIN {X 0,Y 591.946,Z 357.306,A -85,B 0,C 180,E1 26846.903,E2 26846.903} C_VEL
LIN {X 0,Y 592.033,Z 357.304,A -85,B 0,C 180,E1 26843.805,E2 26843.805} C_VEL
LIN {X 0,Y 591.951,Z 357.305,A -85,B 0,C 180,E1 26840.775,E2 26840.775} C_VEL
LIN {X 0,Y 592.03,Z 357.305,A -85,B 0,C 180,E1 26837.697,E2 26837.697} C_VEL
LIN {X 0,Y 591.956,Z 357.304,A -85,B 0,C 180,E1 26834.576,E2 26834.576} C_VEL
LIN {X 0,Y 592.037,Z 357.304,A -85,B 0,C 180,E1 26831.495,E2 26831.495} C_VEL
LIN {X 0,Y 591.961,Z 357.303,A -85,B 0,C 180,E1 26828.352,E2 26828.352} C_VEL
LIN {X 0,Y 592.036,Z 357.302,A -85,B 0,C 180,E1 26825.232,E2 26825.232} C_VEL
LIN {X 0,Y 591.966,Z 357.303,A -85,B 0,C 180,E1 26822.129,E2 26822.129} C_VEL
LIN {X 0,Y 592.037,Z 357.301,A -85,B 0,C 180,E1 26819.032,E2 26819.032} C_VEL
LIN {X 0,Y 591.972,Z 357.303,A -85,B 0,C 180,E1 26815.932,E2 26815.932} C_VEL
LIN {X 0,Y 592.032,Z 357.3,A -85,B 0,C 180,E1 26812.723,E2 26812.723} C_VEL
LIN {X 0,Y 591.979,Z 357.301,A -85,B 0,C 180,E1 26810.047,E2 26810.047} C_VEL
LIN {X 0,Y 590.984,Z 357.431,A -85,B 0,C 180,E1 26809.301,E2 26809.301} C_VEL
LIN {X 0,Y 584.626,Z 358.23,A -85,B 0,C 180,E1 26807.209,E2 26807.209} C_VEL
LIN {X 0,Y 584.1,Z 358.289,A -85,B 0,C 180,E1 26806.664,E2 26806.664} C_VEL
LIN {X 0,Y 584.045,Z 358.29,A -85,B 0,C 180,E1 26803.49,E2 26803.49} C_VEL
LIN {X 0,Y 584.091,Z 358.286,A -85,B 0,C 180,E1 26800.292,E2 26800.292} C_VEL
LIN {X 0,Y 584.057,Z 358.292,A -85,B 0,C 180,E1 26797.132,E2 26797.132} C_VEL
LIN {X 0,Y 584.064,Z 358.287,A -85,B 0,C 180,E1 26793.761,E2 26793.761} C_VEL
LIN {X 0,Y 584.091,Z 358.295,A -85,B 0,C 180,E1 26790.574,E2 26790.574} C_VEL
LIN {X 0,Y 584.056,Z 358.289,A -85,B 0,C 180,E1 26787.367,E2 26787.367} C_VEL
LIN {X 0,Y 584.098,Z 358.291,A -85,B 0,C 180,E1 26784.225,E2 26784.225} C_VEL
LIN {X 0,Y 584.057,Z 358.29,A -85,B 0,C 180,E1 26780.999,E2 26780.999} C_VEL
LIN {X 0,Y 584.096,Z 358.288,A -85,B 0,C 180,E1 26777.829,E2 26777.829} C_VEL
LIN {X 0,Y 584.062,Z 358.29,A -85,B 0,C 180,E1 26774.71,E2 26774.71} C_VEL
LIN {X 0,Y 584.101,Z 358.285,A -85,B 0,C 180,E1 26771.43,E2 26771.43} C_VEL
LIN {X 0,Y 584.095,Z 358.294,A -85,B 0,C 180,E1 26768.053,E2 26768.053} C_VEL
LIN {X 0,Y 584.07,Z 358.287,A -85,B 0,C 180,E1 26764.744,E2 26764.744} C_VEL
LIN {X 0,Y 584.09,Z 358.285,A -85,B 0,C 180,E1 26761.516,E2 26761.516} C_VEL
LIN {X 0,Y 584.07,Z 358.289,A -85,B 0,C 180,E1 26758.303,E2 26758.303} C_VEL
LIN {X 0,Y 584.089,Z 358.285,A -85,B 0,C 180,E1 26755.101,E2 26755.101} C_VEL
LIN {X 0,Y 584.08,Z 358.291,A -85,B 0,C 180,E1 26751.901,E2 26751.901} C_VEL
LIN {X 0,Y 584.094,Z 358.284,A -85,B 0,C 180,E1 26748.563,E2 26748.563} C_VEL
LIN {X 0,Y 584.091,Z 358.291,A -85,B 0,C 180,E1 26745.282,E2 26745.282} C_VEL
LIN {X 0,Y 584.081,Z 358.279,A -85,B 0,C 180,E1 26742.052,E2 26742.052} C_VEL
LIN {X 0,Y 584.079,Z 358.267,A -85,B 0,C 180,E1 26738.86,E2 26738.86} C_VEL
LIN {X 0,Y 584.116,Z 358.436,A -85,B 0,C 180,E1 26737.348,E2 26737.348} C_VEL
LIN {X 0,Y 585.534,Z 361.927,A -85,B 0,C 180,E1 26736.999,E2 26736.999} C_VEL
LIN {X 0,Y 588.914,Z 367.88,A -85,B 0,C 180,E1 26736.641,E2 26736.641} C_VEL
LIN {X 0,Y 588.186,Z 574.245,A -85,B 0,C 180,E1 26733.599,E2 26733.599} C_VEL
LIN {X 0,Y 587.715,Z 710.514,A -85,B 0,C 180,E1 26731.618,E2 26731.618} C_VEL
LIN {X 0,Y 587.466,Z 734.095,A -85,B 0,C 180,E1 26731.082,E2 26731.082} C_VEL
LIN {X 0,Y 587.232,Z 756.194,A -85,B 0,C 180,E1 26730.4,E2 26730.4} C_VEL
LIN {X 0,Y 586.862,Z 778.597,A -85,B 0,C 180,E1 26729.509,E2 26729.509} C_VEL
LIN {X 0,Y 586.54,Z 800.765,A -85,B 0,C 180,E1 26728.435,E2 26728.435} C_VEL
LIN {X 0,Y 586.147,Z 821.72,A -85,B 0,C 180,E1 26727.211,E2 26727.211} C_VEL
LIN {X 0,Y 585.733,Z 843.243,A -85,B 0,C 180,E1 26725.739,E2 26725.739} C_VEL
LIN {X 0,Y 585.411,Z 863.039,A -85,B 0,C 180,E1 26724.165,E2 26724.165} C_VEL
LIN {X 0,Y 585.056,Z 881.816,A -85,B 0,C 180,E1 26722.436,E2 26722.436} C_VEL
LIN {X 0,Y 584.749,Z 899.058,A -85,B 0,C 180,E1 26720.614,E2 26720.614} C_VEL
LIN {X 0,Y 584.534,Z 914.535,A -85,B 0,C 180,E1 26718.753,E2 26718.753} C_VEL
LIN {X 0,Y 584.324,Z 928.525,A -85,B 0,C 180,E1 26716.815,E2 26716.815} C_VEL
LIN {X 0,Y 584.159,Z 941.707,A -85,B 0,C 180,E1 26714.715,E2 26714.715} C_VEL
LIN {X 0,Y 584.058,Z 952.205,A -85,B 0,C 180,E1 26712.771,E2 26712.771} C_VEL
LIN {X 0,Y 583.985,Z 962.178,A -85,B 0,C 180,E1 26710.598,E2 26710.598} C_VEL
LIN {X 0,Y 583.944,Z 969.783,A -85,B 0,C 180,E1 26708.608,E2 26708.608} C_VEL
LIN {X 0,Y 583.899,Z 976.698,A -85,B 0,C 180,E1 26706.366,E2 26706.366} C_VEL
LIN {X 0,Y 583.921,Z 981.28,A -85,B 0,C 180,E1 26704.435,E2 26704.435} C_VEL
LIN {X 0,Y 583.892,Z 985.231,A -85,B 0,C 180,E1 26702.127,E2 26702.127} C_VEL
LIN {X 0,Y 583.883,Z 987.276,A -85,B 0,C 180,E1 26699.996,E2 26699.996} C_VEL
LIN {X 0,Y 583.905,Z 987.968,A -85,B 0,C 180,E1 26697.77,E2 26697.77} C_VEL
LIN {X 0,Y 583.895,Z 987.081,A -85,B 0,C 180,E1 26695.627,E2 26695.627} C_VEL
LIN {X 0,Y 583.883,Z 984.735,A -85,B 0,C 180,E1 26693.42,E2 26693.42} C_VEL
LIN {X 0,Y 583.915,Z 980.947,A -85,B 0,C 180,E1 26691.316,E2 26691.316} C_VEL
LIN {X 0,Y 583.92,Z 975.647,A -85,B 0,C 180,E1 26689.146,E2 26689.146} C_VEL
LIN {X 0,Y 583.941,Z 968.643,A -85,B 0,C 180,E1 26686.982,E2 26686.982} C_VEL
LIN {X 0,Y 584.02,Z 959.961,A -85,B 0,C 180,E1 26684.783,E2 26684.783} C_VEL
LIN {X 0,Y 584.094,Z 949.836,A -85,B 0,C 180,E1 26682.678,E2 26682.678} C_VEL
LIN {X 0,Y 584.22,Z 937.855,A -85,B 0,C 180,E1 26680.545,E2 26680.545} C_VEL
LIN {X 0,Y 584.377,Z 924.595,A -85,B 0,C 180,E1 26678.521,E2 26678.521} C_VEL
LIN {X 0,Y 584.58,Z 909.498,A -85,B 0,C 180,E1 26676.528,E2 26676.528} C_VEL
LIN {X 0,Y 584.858,Z 893.556,A -85,B 0,C 180,E1 26674.682,E2 26674.682} C_VEL
LIN {X 0,Y 585.156,Z 876.024,A -85,B 0,C 180,E1 26672.914,E2 26672.914} C_VEL
LIN {X 0,Y 585.478,Z 857.397,A -85,B 0,C 180,E1 26671.276,E2 26671.276} C_VEL
LIN {X 0,Y 585.879,Z 837.868,A -85,B 0,C 180,E1 26669.777,E2 26669.777} C_VEL
LIN {X 0,Y 586.187,Z 818.104,A -85,B 0,C 180,E1 26668.473,E2 26668.473} C_VEL
LIN {X 0,Y 586.612,Z 796.13,A -85,B 0,C 180,E1 26667.236,E2 26667.236} C_VEL
LIN {X 0,Y 586.922,Z 774.873,A -85,B 0,C 180,E1 26666.237,E2 26666.237} C_VEL
LIN {X 0,Y 587.27,Z 752.001,A -85,B 0,C 180,E1 26665.37,E2 26665.37} C_VEL
LIN {X 0,Y 587.519,Z 730.009,A -85,B 0,C 180,E1 26664.717,E2 26664.717} C_VEL
LIN {X 0,Y 587.729,Z 707.157,A -85,B 0,C 180,E1 26664.235,E2 26664.235} C_VEL
LIN {X 0,Y 588.502,Z 482.353,A -85,B 0,C 180,E1 26660.97,E2 26660.97} C_VEL
LIN {X 0,Y 588.737,Z 367.239,A -85,B 0,C 180,E1 26659.246,E2 26659.246} C_VEL
LIN {X 0,Y 585.061,Z 361.26,A -85,B 0,C 180,E1 26658.845,E2 26658.845} C_VEL
LIN {X 0,Y 584.108,Z 358.454,A -85,B 0,C 180,E1 26658.514,E2 26658.514} C_VEL
LIN {X 0,Y 584.074,Z 358.268,A -85,B 0,C 180,E1 26655.184,E2 26655.184} C_VEL
LIN {X 0,Y 584.087,Z 358.289,A -85,B 0,C 180,E1 26651.955,E2 26651.955} C_VEL
LIN {X 0,Y 584.077,Z 358.29,A -85,B 0,C 180,E1 26648.764,E2 26648.764} C_VEL
LIN {X 0,Y 584.081,Z 358.289,A -85,B 0,C 180,E1 26645.6,E2 26645.6} C_VEL
LIN {X 0,Y 584.09,Z 358.293,A -85,B 0,C 180,E1 26642.355,E2 26642.355} C_VEL
LIN {X 0,Y 584.095,Z 358.285,A -85,B 0,C 180,E1 26639.019,E2 26639.019} C_VEL
LIN {X 0,Y 584.073,Z 358.29,A -85,B 0,C 180,E1 26635.681,E2 26635.681} C_VEL
LIN {X 0,Y 584.093,Z 358.289,A -85,B 0,C 180,E1 26632.426,E2 26632.426} C_VEL
LIN {X 0,Y 584.061,Z 358.289,A -85,B 0,C 180,E1 26629.246,E2 26629.246} C_VEL
LIN {X 0,Y 584.101,Z 358.293,A -85,B 0,C 180,E1 26626.033,E2 26626.033} C_VEL
LIN {X 0,Y 584.064,Z 358.289,A -85,B 0,C 180,E1 26622.794,E2 26622.794} C_VEL
LIN {X 0,Y 584.056,Z 358.293,A -85,B 0,C 180,E1 26619.455,E2 26619.455} C_VEL
LIN {X 0,Y 584.085,Z 358.289,A -85,B 0,C 180,E1 26616.326,E2 26616.326} C_VEL
LIN {X 0,Y 584.037,Z 358.293,A -85,B 0,C 180,E1 26613.12,E2 26613.12} C_VEL
LIN {X 0,Y 584.098,Z 358.289,A -85,B 0,C 180,E1 26610.011,E2 26610.011} C_VEL
LIN {X 0,Y 584.023,Z 358.294,A -85,B 0,C 180,E1 26606.845,E2 26606.845} C_VEL
LIN {X 0,Y 584.089,Z 358.294,A -85,B 0,C 180,E1 26603.735,E2 26603.735} C_VEL
LIN {X 0,Y 584.011,Z 358.296,A -85,B 0,C 180,E1 26600.695,E2 26600.695} C_VEL
LIN {X 0,Y 584.081,Z 358.295,A -85,B 0,C 180,E1 26597.692,E2 26597.692} C_VEL
LIN {X 0,Y 584.018,Z 358.297,A -85,B 0,C 180,E1 26594.584,E2 26594.584} C_VEL
LIN {X 0,Y 584.103,Z 358.372,A -85,B 0,C 180,E1 26591.579,E2 26591.579} C_VEL
LIN {X 0,Y 585.002,Z 361.112,A -85,B 0,C 180,E1 26591.234,E2 26591.234} C_VEL
LIN {X 0,Y 588.044,Z 368.121,A -85,B 0,C 180,E1 26590.472,E2 26590.472} C_VEL
LIN {X 0,Y 587.873,Z 391.476,A -85,B 0,C 180,E1 26588.868,E2 26588.868} C_VEL
LIN {X 0,Y 588.917,Z 397.367,A -85,B 0,C 180,E1 26588.693,E2 26588.693} C_VEL
LIN {X 0,Y 588.188,Z 603.716,A -85,B 0,C 180,E1 26585.651,E2 26585.651} C_VEL
LIN {X 0,Y 587.71,Z 739.568,A -85,B 0,C 180,E1 26583.677,E2 26583.677} C_VEL
LIN {X 0,Y 587.467,Z 763.248,A -85,B 0,C 180,E1 26583.148,E2 26583.148} C_VEL
LIN {X 0,Y 587.253,Z 783.74,A -85,B 0,C 180,E1 26582.526,E2 26582.526} C_VEL
LIN {X 0,Y 586.875,Z 807.109,A -85,B 0,C 180,E1 26581.619,E2 26581.619} C_VEL
LIN {X 0,Y 586.587,Z 828.561,A -85,B 0,C 180,E1 26580.595,E2 26580.595} C_VEL
LIN {X 0,Y 586.172,Z 849.008,A -85,B 0,C 180,E1 26579.425,E2 26579.425} C_VEL
LIN {X 0,Y 585.845,Z 869.343,A -85,B 0,C 180,E1 26578.072,E2 26578.072} C_VEL
LIN {X 0,Y 585.457,Z 888.561,A -85,B 0,C 180,E1 26576.582,E2 26576.582} C_VEL
LIN {X 0,Y 585.096,Z 907.99,A -85,B 0,C 180,E1 26574.85,E2 26574.85} C_VEL
LIN {X 0,Y 584.849,Z 925.079,A -85,B 0,C 180,E1 26573.109,E2 26573.109} C_VEL
LIN {X 0,Y 584.574,Z 941.126,A -85,B 0,C 180,E1 26571.225,E2 26571.225} C_VEL
LIN {X 0,Y 584.345,Z 956.345,A -85,B 0,C 180,E1 26569.177,E2 26569.177} C_VEL
LIN {X 0,Y 584.206,Z 969.632,A -85,B 0,C 180,E1 26567.122,E2 26567.122} C_VEL
LIN {X 0,Y 584.086,Z 980.825,A -85,B 0,C 180,E1 26565.084,E2 26565.084} C_VEL
LIN {X 0,Y 584.009,Z 990.87,A -85,B 0,C 180,E1 26562.963,E2 26562.963} C_VEL
LIN {X 0,Y 583.936,Z 998.686,A -85,B 0,C 180,E1 26560.959,E2 26560.959} C_VEL
LIN {X 0,Y 583.933,Z 1005.469,A -85,B 0,C 180,E1 26558.867,E2 26558.867} C_VEL
LIN {X 0,Y 583.904,Z 1010.835,A -85,B 0,C 180,E1 26556.689,E2 26556.689} C_VEL
LIN {X 0,Y 583.898,Z 1014.59,A -85,B 0,C 180,E1 26554.619,E2 26554.619} C_VEL
LIN {X 0,Y 583.915,Z 1017.053,A -85,B 0,C 180,E1 26552.358,E2 26552.358} C_VEL
LIN {X 0,Y 583.893,Z 1017.939,A -85,B 0,C 180,E1 26550.297,E2 26550.297} C_VEL
LIN {X 0,Y 583.912,Z 1017.325,A -85,B 0,C 180,E1 26548.04,E2 26548.04} C_VEL
LIN {X 0,Y 583.915,Z 1015.28,A -85,B 0,C 180,E1 26545.879,E2 26545.879} C_VEL
LIN {X 0,Y 583.924,Z 1011.466,A -85,B 0,C 180,E1 26543.613,E2 26543.613} C_VEL
LIN {X 0,Y 583.927,Z 1006.557,A -85,B 0,C 180,E1 26541.535,E2 26541.535} C_VEL
LIN {X 0,Y 583.939,Z 999.417,A -85,B 0,C 180,E1 26539.246,E2 26539.246} C_VEL
LIN {X 0,Y 584.008,Z 991.709,A -85,B 0,C 180,E1 26537.244,E2 26537.244} C_VEL
LIN {X 0,Y 584.082,Z 981.374,A -85,B 0,C 180,E1 26535.023,E2 26535.023} C_VEL
LIN {X 0,Y 584.197,Z 970.253,A -85,B 0,C 180,E1 26532.986,E2 26532.986} C_VEL
LIN {X 0,Y 584.337,Z 957.063,A -85,B 0,C 180,E1 26530.928,E2 26530.928} C_VEL
LIN {X 0,Y 584.567,Z 942.57,A -85,B 0,C 180,E1 26528.953,E2 26528.953} C_VEL
LIN {X 0,Y 584.786,Z 927.422,A -85,B 0,C 180,E1 26527.156,E2 26527.156} C_VEL
LIN {X 0,Y 585.066,Z 909.673,A -85,B 0,C 180,E1 26525.312,E2 26525.312} C_VEL
LIN {X 0,Y 585.425,Z 892.25,A -85,B 0,C 180,E1 26523.721,E2 26523.721} C_VEL
LIN {X 0,Y 585.728,Z 873.386,A -85,B 0,C 180,E1 26522.228,E2 26522.228} C_VEL
LIN {X 0,Y 586.143,Z 851.771,A -85,B 0,C 180,E1 26520.748,E2 26520.748} C_VEL
LIN {X 0,Y 586.501,Z 831.912,A -85,B 0,C 180,E1 26519.585,E2 26519.585} C_VEL
LIN {X 0,Y 586.848,Z 810.317,A -85,B 0,C 180,E1 26518.524,E2 26518.524} C_VEL
LIN {X 0,Y 587.15,Z 789.629,A -85,B 0,C 180,E1 26517.68,E2 26517.68} C_VEL
LIN {X 0,Y 587.44,Z 767.026,A -85,B 0,C 180,E1 26516.956,E2 26516.956} C_VEL
LIN {X 0,Y 587.624,Z 746.188,A -85,B 0,C 180,E1 26516.448,E2 26516.448} C_VEL
LIN {X 0,Y 587.818,Z 715.62,A -85,B 0,C 180,E1 26515.955,E2 26515.955} C_VEL
LIN {X 0,Y 588.521,Z 505.303,A -85,B 0,C 180,E1 26512.911,E2 26512.911} C_VEL
LIN {X 0,Y 588.741,Z 395.521,A -85,B 0,C 180,E1 26511.265,E2 26511.265} C_VEL
LIN {X 0,Y 587.759,Z 390.108,A -85,B 0,C 180,E1 26511.06,E2 26511.06} C_VEL
LIN {X 0,Y 587.942,Z 367.546,A -85,B 0,C 180,E1 26509.479,E2 26509.479} C_VEL
LIN {X 0,Y 584.145,Z 358.598,A -85,B 0,C 180,E1 26508.478,E2 26508.478} C_VEL
LIN {X 0,Y 584.023,Z 358.268,A -85,B 0,C 180,E1 26507.696,E2 26507.696} C_VEL
LIN {X 0,Y 584.051,Z 358.287,A -85,B 0,C 180,E1 26504.855,E2 26504.855} C_VEL
LIN {X 0,Y 584.025,Z 358.296,A -85,B 0,C 180,E1 26501.576,E2 26501.576} C_VEL
LIN {X 0,Y 584.046,Z 358.288,A -85,B 0,C 180,E1 26498.672,E2 26498.672} C_VEL
LIN {X 0,Y 584.02,Z 358.286,A -85,B 0,C 180,E1 26495.427,E2 26495.427} C_VEL
LIN {X 0,Y 584.029,Z 358.295,A -85,B 0,C 180,E1 26492.624,E2 26492.624} C_VEL
LIN {X 0,Y 584.018,Z 358.293,A -85,B 0,C 180,E1 26489.317,E2 26489.317} C_VEL
LIN {X 0,Y 584.018,Z 358.295,A -85,B 0,C 180,E1 26486.541,E2 26486.541} C_VEL
LIN {X 0,Y 584.025,Z 358.293,A -85,B 0,C 180,E1 26483.18,E2 26483.18} C_VEL
LIN {X 0,Y 584.026,Z 358.294,A -85,B 0,C 180,E1 26480.336,E2 26480.336} C_VEL
LIN {X 0,Y 584.031,Z 358.293,A -85,B 0,C 180,E1 26477.022,E2 26477.022} C_VEL
LIN {X 0,Y 584.03,Z 358.293,A -85,B 0,C 180,E1 26474.171,E2 26474.171} C_VEL
LIN {X 0,Y 584.036,Z 358.292,A -85,B 0,C 180,E1 26470.854,E2 26470.854} C_VEL
LIN {X 0,Y 584.037,Z 358.293,A -85,B 0,C 180,E1 26467.971,E2 26467.971} C_VEL
LIN {X 0,Y 584.037,Z 358.29,A -85,B 0,C 180,E1 26464.615,E2 26464.615} C_VEL
LIN {X 0,Y 584.052,Z 358.294,A -85,B 0,C 180,E1 26461.667,E2 26461.667} C_VEL
LIN {X 0,Y 584.042,Z 358.29,A -85,B 0,C 180,E1 26458.43,E2 26458.43} C_VEL
LIN {X 0,Y 584.067,Z 358.294,A -85,B 0,C 180,E1 26455.385,E2 26455.385} C_VEL
